// TwinCAT 3 PLC project ContinuousFormulation
// ProgramVersion: 3.1.4020.1
// libraries:
//   VisuElemTextEditor, 3.5.6.0 (System)
//   visuinputs, 3.5.6.0 (system)
//   VisuNativeControl, 3.5.6.0 (System)
//   Tc2_ModbusSrv, * (Beckhoff Automation GmbH)
//   Tc2_SerialCom, * (Beckhoff Automation GmbH)
//   Tc2_Standard, * (Beckhoff Automation GmbH)
//   Tc2_System, * (Beckhoff Automation GmbH)
//   Tc2_SystemCX, * (Beckhoff Automation GmbH)
//   Tc2_Utilities, * (Beckhoff Automation GmbH)
//   Tc3_Interfaces, * (Beckhoff Automation GmbH)
//   Tc3_Module, * (Beckhoff Automation GmbH)
//   VisuDialogs, * (System)
// project tree:
//   DUTs/Wiesler/ ControllerData.TcDUT, elementStatus.TcDUT, FlowCalTestResult.TcDUT, AI.TcDUT, MovingAverage.TcDUT, OLSResult.TcDUT, sAnalogSim.TcDUT, sEU_SCALE.TcDUT, sAnalogConstraint.TcDUT, sWeight.TcDUT, testResults.TcDUT
//   DUTs/Wiesler/Masterflex/ sMasterflexPort.TcDUT
//   / GlobalTextList.TcGTLO, PlcTask.TcTTO
//   GVLs/ Wiesler.TcGVL
//   POUs/FlowCalibration/ FlowCalSequence.TcPOU, OLS.TcPOU, testOLS.TcPOU
//   POUs/ MAIN.TcPOU, MTSerial.TcPOU, sonotecCalibration.TcPOU, FlowCheck.TcPOU, SonotecFreq.TcPOU
//   POUs/Wiesler/ AI1.TcPOU, AO1.TcPOU, fbDatalogger.TcPOU, fbGetUnixTime.TcPOU, fbMovingAverage.TcPOU, FQ1.TcPOU, ModbusTCPReveal.TcPOU, MT_SICS_TO_Weight.TcPOU, randn.TcPOU
//   POUs/Wiesler/DataConversion/ wordArray2Real.TcPOU, wordArray2DINT.TcPOU
//   POUs/Wiesler/Datalog/ fbDatalogger_100ms.TcPOU, fbDatalogger_10ms.TcPOU, fbDatalogger_1ms.TcPOU, fbDatalogger_1s.TcPOU, fbDatalogger_20ms.TcPOU, fShiftArray.TcPOU
//   POUs/Wiesler/FlowConcentrationControl/ CC1.TcPOU, FC2_Preload.TcPOU, FlowSequence_CC1Test.TcPOU, FVC3.TcPOU, StartStopSequence_CC1Test.TcPOU, FV3.TcPOU, testFC.TcPOU (not stored)
//   POUs/Wiesler/Masterflex/ fbMasterflex.TcPOU, fbMasterflexControl.TcPOU, fbMasterflexSerial.TcPOU
//   VISUs/ ContinuousFormulation.TcVIS, HMI.TcVIS, ImagePool.TcIPO (not stored), VisualizationManager.TcVMO (not stored)
// real-time tasks:
//   TASK PlcTask: cycle T#1ms, priority 20, ADS port 350
// I/O:
//   DEVICE Device 1 (EtherCAT), AmsNetId 5.31.160.194.2.1
//     Term 1 (EK1200) [EK1200-5000 EtherCAT Power supply (2A E-Bus)]
//       Term 2 (EL1004) [EL1004 4Ch. Dig. Input 24V, 3ms]
//       Term 3 (EL2004) [EL2004 4Ch. Dig. Output 24V, 0.5A]
//       Term 4 (EL3124) Flow [EL3124 4Ch. Ana. Input 4-20mA Diff.]
//       Term 5 (EL3124) Optek [EL3124 4Ch. Ana. Input 4-20mA Diff.]
//       Term 6 (EL3124) Reveal [EL3124 4Ch. Ana. Input 4-20mA Diff.]
//       Term 7 (EL3124) [EL3124 4Ch. Ana. Input 4-20mA Diff.]
//       Term 8 (EL3104) [EL3104 4Ch. Ana. Input +/-10V Diff.]
//       Term 9 (EL3702) [EL3702 2Ch. Ana. Input +/-10V, DIFF, Oversample]
//       Term 10 (EL4124) [EL4124 4Ch. Ana. Output 4-20mA, 16bit]
//       Term 11 (EL6002) [EL6002 Interface 2Ch. (RS232)]
//       Term 12 (EL6002) [EL6002 Interface 2Ch. (RS232)]
//       Term 13 (EL1502) [EL1502 2Ch. +/- Counter 24V, 100kHz]
//       Term 14 (EL9011) [EL9011 End Terminal]
// variable links:
//   ContinuousFormulation/ContinuousFormulation Instance <-> Device 1 (EtherCAT)/Term 1 (EK1200)/Term 11 (EL6002)
//     PlcTask Inputs/MAIN.P9999A.stIn_Port/D[{0..21}] <-> COM TxPDO-Map Inputs Channel 1/Data In {0..21}  (22 links)
//     PlcTask Inputs/MAIN.P9999A.stIn_Port/Status <-> COM TxPDO-Map Inputs Channel 1/Status
//     PlcTask Inputs/MAIN.P9999B.stIn_Port/D[{0..21}] <-> COM TxPDO-Map Inputs Channel 2/Data In {0..21}  (22 links)
//     PlcTask Inputs/MAIN.P9999B.stIn_Port/Status <-> COM TxPDO-Map Inputs Channel 2/Status
//     PlcTask Outputs/MAIN.P9999A.stOut_Port/Ctrl <-> COM RxPDO-Map Outputs Channel 1/Ctrl
//     PlcTask Outputs/MAIN.P9999A.stOut_Port/D[{0..21}] <-> COM RxPDO-Map Outputs Channel 1/Data Out {0..21}  (22 links)
//     PlcTask Outputs/MAIN.P9999B.stOut_Port/Ctrl <-> COM RxPDO-Map Outputs Channel 2/Ctrl
//     PlcTask Outputs/MAIN.P9999B.stOut_Port/D[{0..21}] <-> COM RxPDO-Map Outputs Channel 2/Data Out {0..21}  (22 links)
//   ContinuousFormulation/ContinuousFormulation Instance <-> Device 1 (EtherCAT)/Term 1 (EK1200)/Term 12 (EL6002)
//     PlcTask Inputs/MTSerial.stIn_Port/D[{0..21}] <-> COM TxPDO-Map Inputs Channel 1/Data In {0..21}  (22 links)
//     PlcTask Inputs/MTSerial.stIn_Port/Status <-> COM TxPDO-Map Inputs Channel 1/Status
//     PlcTask Outputs/MTSerial.stOut_Port/Ctrl <-> COM RxPDO-Map Outputs Channel 1/Ctrl
//     PlcTask Outputs/MTSerial.stOut_Port/D[{0..21}] <-> COM RxPDO-Map Outputs Channel 1/Data Out {0..21}  (22 links)
//   ContinuousFormulation/ContinuousFormulation Instance <-> Device 1 (EtherCAT)/Term 1 (EK1200)/Term 2 (EL1004)
//     PlcTask Inputs/MAIN.AC9999C.lsh <-> Channel 2/Input
//     PlcTask Inputs/MAIN.AC9999C.lsl <-> Channel 1/Input
//   ContinuousFormulation/ContinuousFormulation Instance <-> Device 1 (EtherCAT)/Term 1 (EK1200)/Term 3 (EL2004)
//     PlcTask Outputs/MAIN.FV9999C.activeSV <-> Channel 2/Output
//     PlcTask Outputs/MAIN.FV9999C.passiveSV <-> Channel 1/Output
//   ContinuousFormulation/ContinuousFormulation Instance <-> Device 1 (EtherCAT)/Term 1 (EK1200)/Term 4 (EL3124) Flow
//     PlcTask Inputs/MAIN.FT9999A.raw <-> AI Standard Channel 2/Value
//     PlcTask Inputs/MAIN.FT9999A.status <-> AI Standard Channel 2/Status
//     PlcTask Inputs/MAIN.FT9999B.raw <-> AI Standard Channel 1/Value
//     PlcTask Inputs/MAIN.FT9999B.status <-> AI Standard Channel 1/Status
//     PlcTask Inputs/MAIN.FT9999C.raw <-> AI Standard Channel 3/Value
//     PlcTask Inputs/MAIN.FT9999C.status <-> AI Standard Channel 3/Status
//   ContinuousFormulation/ContinuousFormulation Instance <-> Device 1 (EtherCAT)/Term 1 (EK1200)/Term 6 (EL3124) Reveal
//     PlcTask Inputs/MAIN.AT9999RV{290..320 step 10}.raw <-> AI Standard Channel {1..4}/Value  (4 links)
//     PlcTask Inputs/MAIN.AT9999RV{290..320 step 10}.status <-> AI Standard Channel {1..4}/Status  (4 links)
//   ContinuousFormulation/ContinuousFormulation Instance <-> Device 1 (EtherCAT)/Term 1 (EK1200)/Term 8 (EL3104)
//     PlcTask Inputs/MAIN.AT9999CWx.raw <-> AI Standard Channel 4/Value
//     PlcTask Inputs/MAIN.AT9999CWx.status <-> AI Standard Channel 4/Status
//     PlcTask Inputs/MAIN.PT9999A.raw <-> AI Standard Channel 1/Value
//     PlcTask Inputs/MAIN.PT9999A.status <-> AI Standard Channel 1/Status
//     PlcTask Inputs/MAIN.PT9999B.raw <-> AI Standard Channel 2/Value
//     PlcTask Inputs/MAIN.PT9999B.status <-> AI Standard Channel 2/Status
//     PlcTask Inputs/MAIN.PT9999C.raw <-> AI Standard Channel 3/Value
//     PlcTask Inputs/MAIN.PT9999C.status <-> AI Standard Channel 3/Status
//   ContinuousFormulation/ContinuousFormulation Instance <-> Device 1 (EtherCAT)/Term 1 (EK1200)/Term 9 (EL3702)
//     PlcTask Inputs/MAIN.AT9999CWYY.raw <-> Ch2 Sample 0/Ch2 Value
//     PlcTask Inputs/MAIN.AT9999CWy.raw <-> Ch1 Sample 0/Ch1 Value

CONFIGURATION ContinuousFormulation
    RESOURCE PLC ON TwinCAT3
        TASK PlcTask(INTERVAL := T#1ms, PRIORITY := 20);
        PROGRAM MAIN WITH PlcTask : MAIN;
        PROGRAM FlowCheck WITH PlcTask : FlowCheck;
        PROGRAM StartStopSequence_CC1Test WITH PlcTask : StartStopSequence_CC1Test;
    END_RESOURCE
END_CONFIGURATION

// ---- DUTs/Wiesler/ControllerData.TcDUT
TYPE ControllerData :
STRUCT
	Kp : LREAL := 1.0; //Gain
	Ti : TIME := T#5S; //Integral time
	execTime : TIME := T#500MS; //Time between controller executions
END_STRUCT
END_TYPE

// ---- DUTs/Wiesler/elementStatus.TcDUT
TYPE elementStatus :
(
    Bad := 0,
    Timeout := 1,
	Unknown := 11,
    Good := 12
);
END_TYPE

// ---- DUTs/Wiesler/FlowCalTestResult.TcDUT
TYPE FlowCalTestResult :
STRUCT
	flow : LREAL;
	weight : LREAL;
	startTime : 
END_STRUCT
END_TYPE

// ---- DUTs/Wiesler/Masterflex/sMasterflexPort.TcDUT
TYPE sMasterflexPort :
STRUCT
	// I/O variables for a EL6001 terminal
	stIn_Port AT %I*	: EL6inData22B;	// linked to the EL6002 in the TwinCAT System Manager
	stOut_Port AT %Q*	: EL6outData22B; // linked to the EL6002 in the TwinCAT System Manager
	
	//Serial send variables
	sSendString: STRING(100) := '';

	//Receive variables
	bReceiveTimeout	: BOOL := FALSE;
	sRxSuffix : STRING(5) := '';
	nReceiveCounter	: UDINT := 0;
	sLastReceivedString: STRING(30) := '';
	bListening : BOOL := FALSE;
	tListenTON : TON;
	
	//Pump Status
	fSpeedPV : LREAL := -100.0;
	fFlowPV : LREAL := 0.0;		//Calculated flow in mg/min
	fSpeedSP : LREAL := -100.0;
	fFlowSP : LREAL := -100.0;
	bRun : BOOL := FALSE;
	bLocal : BOOL := FALSE;
	bDirection : BOOL := TRUE; //true is positive/forward, false is negative/backwards
	nPumpStatus : INT := -1; //see http://www.coleparmer.com/Assets/manual_pdfs/07551-20,30.pdf pg 3-33
	nCommStatus : INT := -1;
	
	//Pump Requests
	fSpeedSP_RQ : LREAL := 0.0;
	fFlowSP_RQ : LREAL := -100.0;
	nRun_RQ : INT := 0;  //-1=no RQ, 0=Stop, 1=Run
	nDir_RQ : INT := -1;  //-1=no RQ, 0=Backwards, 1=Forwards //TODO this does no twork correctly probably. Pump must be stopped to change direction
	nLocal_RQ : INT := 1; //-1=no RQ, 0=Remote, 1=Local

	//State Control Information
	nLastState : INT := 1;
	nState : INT := 1;
	
	//Pump Configuration
	//Tube Sizes: 13 (.8mm, 1/32"), 14 (1.6mm, 1/16"), 16 (3.1mm, 1/8"), 
	//			  25 (4.8mm, 3/16"), 17 (6.4mm, 1/4"), 18 (7.9mm, 5/16")
	nTubeSize :INT := 13;		//Tube Number
	nHeads : INT := 2;			//Number of heads
	fPeriodMS : LREAL := 1.0;	//Period between pulses in milliseconds
	
	
END_STRUCT
END_TYPE

// ---- DUTs/Wiesler/AI.TcDUT
TYPE AI :
STRUCT
	// IO variables: status and value
	raw AT %I* : INT;
	status AT %I* : INT;
	// AI scaling and simulation
	scale : sEU_SCALE := (euLo := 0,  euHi := 100.0, eu := 'mg/min');
	sim : sAnalogSim;
	// PV and filtered PV
	pv : LREAL := -1000.0;
	pvfilt : LREAL := -1000.0;
	//Low cutoff 
	loCutEnable : BOOL := FALSE; //low cutoff enable
	loCut : LREAL := 0.0; // if pv is less than this, set pv to 0.0
END_STRUCT
END_TYPE

// ---- DUTs/Wiesler/MovingAverage.TcDUT
TYPE MovingAverage :
STRUCT
	arrSize : UINT := 3000; //Do not change online.
	start : UINT := arrSize - 1;
	vals : ARRAY[0..start] OF LREAL := [arrSize(0.0)];
	size : UINT := 1000;
	in : LREAL;
	out : LREAL;
END_STRUCT
END_TYPE

// ---- DUTs/Wiesler/OLSResult.TcDUT
TYPE OLSResult :
STRUCT
	m : LREAL := 0; // calculated linear regression slope
	b : LREAL := 0; // calculated linear regression intercept
	R2 : LREAL := 0; // R squared
	status : INT := 0; // 0 : OK; >0 : any failure
END_STRUCT
END_TYPE

// ---- DUTs/Wiesler/sAnalogSim.TcDUT
TYPE sAnalogSim :
STRUCT
	simEnable : BOOL := FALSE;
	simValue : LREAL := 0.0;
END_STRUCT
END_TYPE

// ---- DUTs/Wiesler/sEU_SCALE.TcDUT
TYPE sEU_SCALE :
STRUCT
	rawLo: INT := 0;
	rawHi: INT := 32767;
	euLo: LREAL := 0.0;
	euHi: LREAL := 100.0;
	eu: STRING[20] := '%';
END_STRUCT
END_TYPE

// ---- DUTs/Wiesler/sAnalogConstraint.TcDUT
TYPE sAnalogConstraint :
STRUCT
	sp : LREAL := 0.0;  //value to be sent to controller
	rq : LREAL := 0.0;  //request from HMI or calculations
	mn : LREAL := 0.0;  //Minimum value
	mx : LREAL := 0.0;  //Maximum value
END_STRUCT
END_TYPE

// ---- DUTs/Wiesler/sWeight.TcDUT
TYPE sWeight :
STRUCT
	pv : LREAL := -10000.0;
	status : string(15) := 'Invalid';
END_STRUCT
END_TYPE

// ---- DUTs/Wiesler/testResults.TcDUT
TYPE testResults :
STRUCT
	P9999Arpm : LREAL := 0.0;
	P9999Atubing : INT := 0;
	P9999Brpm : LREAL := 0.0;
	P9999Btubing : INT := 0;
	FQ9999A : LREAL := 0.0;
	FQ9999B : LREAL := 0.0;
	FQ9999C : LREAL := 0.0;
	FT9999Aavg : LREAL := 0.0;
	FT9999Bavg : LREAL := 0.0;
	FT9999Cavg : LREAL := 0.0;
END_STRUCT
END_TYPE

// ---- GVLs/Wiesler.TcGVL
VAR_GLOBAL
	unixTime : ULINT;
	FC9999ACtrlData : ControllerData := (Kp := 7.0, Ti := T#500MS, execTime := T#200MS);
	FC9999BCtrlData : ControllerData := (Kp := 0.4, Ti := T#500MS, execTime := T#500MS);
END_VAR

VAR_GLOBAL PERSISTENT
	FT9999A_OLS : OLSResult := (m := 1.0, b := 0.0, R2 := 1.0, status := 0);
	P9999A_OLS : OLSResult := (m := 1.0, b := 0.0, R2 := 1.0, status := 0);
	FT9999B_OLS : OLSResult := (m := 1.0, b := 0.0, R2 := 1.0, status := 0);
	P9999B_OLS : OLSResult := (m := 1.0, b := 0.0, R2 := 1.0, status := 0);
END_VAR

// ---- POUs/MAIN.TcPOU
PROGRAM MAIN

VAR CONSTANT
	SAMPLE_SIZE : INT := 1000;
END_VAR

VAR_INPUT
	logActive : BOOL := FALSE;
	MTSendString : STRING(132) := 'SIR$0D$0A';
	//Pump control
	P9999A : sMasterflexPort := (bDirection := FALSE, nTubeSize := 13);
	P9999B : sMasterflexPort := (bDirection := FALSE, nTubeSize := 16);
	//totalizer blocks
	fbFQ9999A : FQ1;
	fbFQ9999B : FQ1;
	fbFQ9999C : FQ1;
	FQ9999_MasterReset : BOOL; //Master reset - resets all totalizers
	AQ9999C : LREAL; // implied concentration based on FQA and FQB
	
	phase : UINT := 0;
	//Flow and Concentration Control
	FC9999A : FC2_Preload;
	FC9999B : FC2_Preload;
	AC9999C : CC1;
	FV9999C : FV3;
	FVC9999C : FVC3;

END_VAR

VAR
	//test
    Tau : LREAL := 1.0;
	FilterFactor : LREAL;
	ftfirstorder : LREAL;
	//-test
	heartbeat : DINT;
	fbGetUnixTimeGlobal : fbGetUnixTime;
	temp : UINT;
	MTWeight : sWeight;
	
	//Flowmeters
	FT9999A : AI := (loCutEnable:= FALSE, loCut := 0.25, scale := (euLo := -20.0,  euHi := 100.0, eu := 'ml/min')); //E+H small
	FT9999B : AI := (loCutEnable:= TRUE, loCut := 2.25, scale := (euLo := 0,  euHi := 1000.0, eu := 'ml/min')); //E+H large
	FT9999C : AI := (loCutEnable:= TRUE, loCut := 2.25, scale := (euLo := 0,  euHi := 1000.0, eu := 'ml/min')); //E+H very large
	
	//Pressures
	PT9999A : AI := (scale := (euLo := 0,  euHi := 15.0, eu := 'psig'));
	PT9999B : AI := (scale := (euLo := 0,  euHi := 15.0, eu := 'psig'));
	PT9999C : AI := (scale := (euLo := 0,  euHi := 15.0, eu := 'psig'));

	//Reveal
	AT9999RV290 : AI := (scale := (euLo := -0.1,  euHi := 2.0, eu := 'AU'));
	AT9999RV300 : AI := (scale := (euLo := -0.1,  euHi := 1.1, eu := 'mg/ml'));
	AT9999RV310 : AI := (scale := (euLo := 0,  euHi := 2.0, eu := 'AU'));
	AT9999RV320 : AI := (scale := (euLo := 0,  euHi := 2.0, eu := 'AU'));
	AT9999C : ModbusTCPReveal();

	//ColorWise
	AT9999CWx  : AI := (scale := (rawLo := 0, rawHi := 16383, euLo := 0,  euHi := 1.0, eu := 'x'));
	AT9999CWy  : AI := (scale := (rawLo := 0, rawHi := 16383, euLo := 0,  euHi := 1.0, eu := 'y'));
	AT9999CWYY : AI := (scale := (rawLo := 0, rawHi := 16383, euLo := 0,  euHi := 1.0, eu := 'Y'));

	//function blocks
	fbP9999A : fbMasterflex;
	fbP9999B : fbMasterflex;
	
	//Phases
	FT9999A_FLOWCAL : FlowCalSequence;
	FT9999B_FLOWCAL : FlowCalSequence;
	
	//AI blocks
	fbFT9999A : AI1;
	fbFT9999B : AI1;
	fbFT9999C : AI1;
	fbPT9999A : AI1;
	fbPT9999B : AI1;
	fbPT9999C : AI1;
	fbAT9999RV290 : AI1;
	fbAT9999RV300 : AI1;
	fbAT9999RV310 : AI1;
	fbAT9999RV320 : AI1;
	fbAT9999CWx  : AI1;
	fbAT9999CWy  : AI1;
	fbAT9999CWYY : AI1;
	
	// filter blocks
	fbFT9999AFilt : fbMovingAverage;
	FT9999ASize : UINT := 500;
	FT9999AFiltTarget : LREAL := 1500.0; //Target number of ms to for moving average
	fbFT9999BFilt : fbMovingAverage;
	FT9999BSize : UINT := 500;
	FT9999BFiltTarget : LREAL := 1500.0; //Target number of ms to for moving average
	fbFT9999CFilt : fbMovingAverage;
	FT9999CSize : UINT := 500;
	fbFT9999CfqFilt : fbMovingAverage;

	//Data logging
	fbP9999ARPMlog : fbDatalogger_100ms;
	fbP9999AFlowlog : fbDatalogger_100ms;
	fbP9999BRPMlog : fbDatalogger_100ms;
	fbP9999BFlowlog : fbDatalogger_100ms;
		
	fbFT9999Alog : fbDatalogger_1ms;
	fbFT9999Blog : fbDatalogger_1ms;
	fbFT9999Clog : fbDatalogger_1ms;
	
	fbFT9999Afiltlog : fbDatalogger_100ms;
	fbFT9999Bfiltlog : fbDatalogger_100ms;
	fbFT9999Cfiltlog : fbDatalogger_100ms;
	
	fbFQ9999Alog : fbDatalogger_100ms;
	fbFQ9999Blog : fbDatalogger_100ms;
	fbFQ9999Clog : fbDatalogger_100ms;
	
	fbPT9999Alog : fbDatalogger_1ms;
	fbPT9999Blog : fbDatalogger_1ms;
	fbPT9999Clog : fbDatalogger_1ms;

	fbWT9999Clog : fbDatalogger_100ms;

	fbAT9999RV290log : fbDatalogger_10ms;
	fbAT9999RV300log : fbDatalogger_10ms;
	fbAT9999RV310log : fbDatalogger_10ms;
	fbAT9999RV320log : fbDatalogger_10ms;

	fbAT9999CWxlog  : fbDatalogger_1ms;
	fbAT9999CWylog  : fbDatalogger_1ms;
	fbAT9999CWYYlog : fbDatalogger_1ms;
	
END_VAR

heartbeat := heartbeat + 1;
fbGetUnixTimeGlobal();  //set global variable unixTime
//Code that runs 1 time per second
IF (heartbeat MOD 1000) = 0 THEN
	temp := MIN(2499,DINT_TO_UINT(3*TRUNC(P9999A.fPeriodMS)));  //lower bound is 3 * period - want to make sure at least 3 periods are averaged
	FT9999ASize := LIMIT(temp, DINT_TO_UINT((TRUNC(P9999A.fPeriodMS) * TRUNC(FT9999AFiltTarget/P9999A.fPeriodMS))), 2500);
	temp := MIN(2499,DINT_TO_UINT(3*TRUNC(P9999B.fPeriodMS)));  //lower bound is 3 * period - want to make sure at least 3 periods are averaged
	FT9999BSize := LIMIT(temp, DINT_TO_UINT((TRUNC(P9999B.fPeriodMS) * TRUNC(FT9999BFiltTarget/P9999B.fPeriodMS))), 2500);
END_IF

//Call serial line handlers
MTSerial(sSendString := MTSendString, weight := MTWeight);

//Call pump handler
fbP9999A(sPort := P9999A);
fbP9999B(sPort := P9999B);

//Valve handlers
fv9999c();


//Flow transmitters
fbFT9999A(AI := FT9999A);
fbFT9999AFilt(in := FT9999A.pv, size := FT9999ASize, out => FT9999A.pvfilt);

//test
FilterFactor := 1.0 - EXP(-0.001/tau);
ftfirstorder := (1.0 - filterfactor) * ftfirstorder + filterfactor * FT9999A.pv;
//-test


fbFQ9999A(flow := FT9999A.pv, timeBaseMS := (1000.0*60.0));
fbFT9999B(AI := FT9999B);
fbFT9999BFilt(in := FT9999B.pv, size := FT9999BSize, out => FT9999B.pvfilt);
fbFQ9999B(flow := FT9999B.pv, timeBaseMS := (1000.0*60.0));
fbFT9999C(AI := FT9999C);
fbFT9999CFilt(in := FT9999C.pv, size := FT9999CSize, out => FT9999C.pvfilt);
fbFQ9999C(flow := FT9999C.pv, timeBaseMS := (1000.0*60.0));
//reset all totalizers if master reset 
IF FQ9999_MasterReset THEN
	fbFQ9999A.resetRQ := TRUE;
	fbFQ9999B.resetRQ := TRUE;
	fbFQ9999C.resetRQ := TRUE;
	FQ9999_MasterReset := FALSE;
END_IF
//Calculate average concentration
IF (fbFQ9999A.total + fbFQ9999B.total) > 0.0 THEN
	AQ9999C := (fbFQ9999A.total*AC9999C.API_Concentration)/(fbFQ9999A.total + fbFQ9999B.total);
ELSE
	AQ9999C := 0.0;
END_IF

//Flow and Concentration Control
FC9999A(FTOLS := FT9999A_OLS, pumpOLS := P9999A_OLS, pump := P9999A, ft := FT9999A, ctrlData:= FC9999ACtrlData);
FC9999B(FTOLS := FT9999B_OLS, pumpOLS := P9999B_OLS, pump := P9999B, ft := FT9999B, ctrlData:= FC9999BCtrlData);
FT9999A_FLOWCAL(fq := fbFQ9999A, pump := P9999A, FTOLS := FT9999A_OLS, pumpOLS := P9999A_OLS);
FT9999B_FLOWCAL(fq := fbFQ9999B, pump := P9999B, FTOLS := FT9999B_OLS, pumpOLS := P9999B_OLS);
AC9999C(FCA := FC9999A, FTA := FT9999A, FCB:= FC9999B, FTB := FT9999B, PumpA := P9999A, PumpB := P9999B);
FVC9999C(FTA := FT9999A, FTB := FT9999B, ATC := AT9999C, cc := AC9999C, API_Concentration := AC9999C.API_Concentration, FV := FV9999C);

//Pressure
fbPT9999A(AI := PT9999A);
fbPT9999B(AI := PT9999B);
fbPT9999C(AI := PT9999C);

//Reveal
AT9999C();

//ColorWise
fbAT9999CWx(AI := AT9999CWx);
fbAT9999CWy(AI := AT9999CWy);
fbAT9999CWYY(AI := AT9999CWYY);

//Data Logging
fbP9999ARPMlog(fData := P9999A.fSpeedPV);
fbP9999AFlowlog(fData := P9999A.fFlowPV);
fbP9999BRPMlog(fData := P9999B.fSpeedPV);
fbP9999BFlowlog(fData := P9999B.fFlowPV);
	
fbFT9999Alog(fData := FT9999A.pv);;
fbFT9999Blog(fData := FT9999B.pv);
fbFT9999Clog(fData := FT9999C.pv);

fbFT9999Afiltlog(fData := FT9999A.pvfilt);
fbFT9999Bfiltlog(fData := FT9999B.pvfilt);
fbFT9999Cfiltlog(fData := FT9999C.pvfilt);

fbFQ9999Alog(fData := fbFQ9999A.total);
fbFQ9999Blog(fData := fbFQ9999B.total);
fbFQ9999Clog(fData := fbFQ9999C.total);

fbPT9999Alog(fData := PT9999A.pv);
fbPT9999Blog(fData := PT9999B.pv);
fbPT9999Clog(fData := PT9999C.pv);

fbWT9999Clog(fData := MTWeight.pv);

fbAT9999RV290log(fData := AT9999RV290.pv);
fbAT9999RV300log(fData := AT9999RV300.pv);
fbAT9999RV310log(fData := AT9999RV310.pv);
fbAT9999RV320log(fData := AT9999RV320.pv);

fbAT9999CWxlog(fData := AT9999CWx.pv);
fbAT9999CWylog(fData := AT9999CWy.pv);
fbAT9999CWYYlog(fData := AT9999CWYY.pv);

//Phase Control
CASE phase OF
1:
	FT9999A_FLOWCAL.start := TRUE;
	phase := 0;
2:
	FT9999B_FLOWCAL.start := TRUE;
	phase := 0;
END_CASE

END_PROGRAM

// ---- POUs/Wiesler/FQ1.TcPOU
FUNCTION_BLOCK FQ1
VAR_INPUT
	enable : BOOL := TRUE;
	resetRQ : BOOL := FALSE;
	flow : LREAL := 0.0;
	timeBaseMS : LREAL := 1000.0*60.0;
END_VAR
VAR_IN_OUT
END_VAR
VAR_OUTPUT
	total : LREAL := 0.0;
END_VAR
VAR
	scanMS : LREAL := 1.0;
END_VAR

IF resetRQ THEN
	total := 0.0;
	resetRQ := FALSE;
ELSE
	IF enable THEN
		total := total + flow*scanMS/timeBaseMS;		
	END_IF
END_IF

END_FUNCTION_BLOCK

// ---- POUs/Wiesler/FlowConcentrationControl/FC2_Preload.TcPOU
FUNCTION_BLOCK FC2_Preload
VAR_INPUT
	SP : LREAL := 0.0;
	uncalFTPV : LREAL := 0;
	modeSP : UINT := 1; //controller mode Setpoint.  1 is Manual, 2 is Auto
	outMax : LREAL := 600.0;
	outMin : LREAL := 10.0; //don't allow pump speed to go below 10 RPM
	SPMin : LREAL := 1.0; //don't allow SP to be less than 1.0 mL/min
END_VAR
VAR_IN_OUT
	FTOLS : OLSResult;
	pumpOLS : OLSResult;
	pump : sMasterflexPort;
	ft : AI;
	ctrlData : ControllerData;
END_VAR
VAR_OUTPUT

END_VAR
VAR
	PV : LREAL := 0.0;
	outBase : LREAL := 0.0 ; //Base OUT value predicted by flow vs. speed correlation
	OUT : LREAL := 0.0;
	lastOUT: LREAL := 0.0;
	modeAct : UINT := 2; //controller mode Actual.  1 is Manual, 2 is Auto, 3 is Suspend
	lastModeAct : UINT;
	execCounter : DWORD := 0;
	iError : LREAL;
	integral : LREAL;
	integralAtOutMax : LREAL;
	integralAtOutMin : LREAL;
	lastIntegral : LREAL;
	lastSP : LREAL;
	
	fbSuspend : TP;
	newSP : BOOL;
	newPumpOn : BOOL;
	pumpModeOn : BOOL;
	lastPumpModeOn : BOOL;
	suspendTime : TIME := T#2S;
	
END_VAR

//PV := FTOLS.m * ft.pvfilt + FTOLS.b;  //DO NOT scale ft to adjust for zero
PV := ft.pvfilt;
SP := MAX(SP, SPMin);
pumpModeOn := ((NOT pump.bLocal AND pump.bRun));
execCounter := execCounter + 1;

modeAct := modeSP;
//Calculate integration suspend - when SP changes or the mode has just gone to Auto.
newSP := (lastSP <> SP OR (modeAct = 2 AND lastModeAct <> 2));
newPumpOn := (lastPumpModeOn <> pumpModeOn);
IF newSP THEN
	//lastIntegral := lastIntegral * SP/MAX(lastSP, 0.01);
	//lastIntegral := LIMIT(outMin, lastIntegral, outMax);
END_IF
fbSuspend(IN := (newSP OR newPumpOn), PT := suspendTime);

//Control algorithm
IF execCounter >= TIME_TO_DWORD(ctrlData.execTime) THEN
	execCounter := 0;
	//Execute control algorithm
	CASE modeAct OF
		2: //Control is in Auto
			outBase := pumpOLS.m * SP + pumpOLS.b;
			//calculate new integral component unless integration is suspended
			IF fbSuspend.Q OR ((modeSP = 2) AND (pump.bLocal OR NOT pump.bRun)) THEN
				iError := 0.0;
			ELSE
				iError := (SP - PV) * ctrlData.Kp * DWORD_TO_LREAL(TIME_TO_DWORD(ctrlData.execTime))/DWORD_TO_LREAL(TIME_TO_DWORD(ctrlData.Ti));
			END_IF		
			//calculate integral taking into account the ARW and Output min and max
			integralAtOutMax := (outMax - outBase);  //integral value that would make OUT = outMax
			integralAtOutMin := (outMin - outBase);  //integral value that would make OUT = outMin
			integral := MAX(integralAtOutMin, MIN(integralAtOutMax,(lastIntegral + iError)));
			//set output to be the bias calculated by the flow vs. speed correlation and integral action
			OUT := outBase + integral;
			OUT := DINT_TO_LREAL(LREAL_TO_DINT(OUT*10.0))/10.0; //round to tenth
			IF OUT <> lastOut THEN
				pump.fSpeedSP_RQ := OUT;
			END_IF
		1: //Control is in Manual
			integral := 0.0;
			OUT := 0.0;		
	END_CASE
	lastIntegral := integral;
	lastOut := OUT;
END_IF

lastSP := SP;
lastPumpModeOn := pumpModeOn;
lastModeAct := modeAct;

END_FUNCTION_BLOCK

// ---- POUs/Wiesler/FlowConcentrationControl/CC1.TcPOU
FUNCTION_BLOCK CC1
//Concentration Control
//Sets FC Setpoints to achieve target concentration.  At this point no feedback.
VAR_INPUT
	mode : UINT := 0; //0 = manual, 1=Final conc and total flow set directly
	API_Concentration : LREAL := 42.0; //	API Concentration in mg/mL
	conc : sAnalogConstraint := (sp := 0.0, rq := -100.0, mn := 0.0, mx := 1.0);
	a : sAnalogConstraint := (sp := 0.0, rq := -100.0, mn := 2.0, mx := 70.0);
	b : sAnalogConstraint := (sp := 0.0, rq := -100.0, mn := 20.0, mx := 500.0);
	c : sAnalogConstraint := (sp := 0.0, rq := -100.0, mn := 0.0, mx := 500.0);
	lsh AT %I* : BOOL := FALSE;
	lsl AT %I* : BOOL := FALSE;
	autoFill : UINT := 0; //0 = manual (not filling), 1 = auto fill ON
END_VAR
VAR_IN_OUT
	FCA : FC2_Preload;
	FTA : AI;
	FCB : FC2_Preload;
	FTB : AI;
	PumpA : sMasterflexPort;
	PumpB : sMasterflexPort;	
END_VAR
VAR_OUTPUT
END_VAR
VAR
	lastMode : UINT := 0;
	lastAPI_Concentration : LREAL := 42.0;
	filling : BOOL := TRUE;
END_VAR

//Determine constraints on concentration and final flow
c.mx := a.mx + b.mx;
c.mn := 0.0;
conc.mx := API_Concentration;
conc.mn := 0.0;
c.sp := LIMIT(c.mn, c.sp, c.mx);
conc.sp := LIMIT(conc.mn, conc.sp, conc.mx);

//Check of concentration or flow requests are different or filling and pumps OFF
IF c.rq <> c.sp OR conc.rq <> conc.sp OR API_Concentration <> lastAPI_Concentration OR (filling AND (NOT PumpA.bRun AND NOT PumpB.bRun)) THEN
	a.rq := c.rq * conc.rq/MAX(0.0001,API_Concentration);
	b.rq := c.rq - a.rq;
	
	//Check if both flows are in valid ranges
	IF (a.rq = 0.0 OR (a.rq >= a.mn AND a.rq <= a.mx)) AND 
       (b.rq = 0.0 OR (b.rq >= b.mn AND b.rq <= b.mx)) THEN
		a.sp := a.rq;
		b.sp := b.rq;
		c.sp := c.rq;
		conc.sp := conc.rq;
	ELSE
		IF API_Concentration <> lastAPI_Concentration THEN //API concetration changed outside acceptable range.  Go to manual
			mode := 0;
		END_IF
		c.rq := c.sp;
		conc.rq := conc.sp;		
	END_IF
END_IF

// check level
IF NOT lsl THEN
	filling := TRUE;
END_IF
IF lsh THEN
	filling := FALSE;
END_IF

IF NOT filling AND autoFill = 1 THEN // if we are NOT filling (and in autoFill mode) then turn off pumps
	a.sp := 0;
	b.sp := 0;
END_IF

//set flow control setpoint and pump on/off command for API and buffer (both have to be on or both off)
//drive pumps and speed setpoints
IF mode = 1 AND (lastMode <> 1 OR ((PumpA.bLocal = TRUE OR PumpB.bLocal=TRUE) AND filling)) THEN
	PumpA.nLocal_RQ := 0;
	PumpB.nLocal_RQ := 0;
END_IF
IF mode = 1 THEN  //only set flow rates and pump states if in Auto and filling (Not discharging)
	//turn on or off pump A
	IF a.sp >= a.mn THEN
		FCA.modeSP := 2; //auto
		FCA.SP := a.sp;
		IF NOT PumpA.bRun THEN
			PumpA.nRun_RQ := 1;
		END_IF
	ELSE
		FCA.modeSP := 1; //manual
		IF PumpA.bRun THEN
			PumpA.nRun_RQ := 0;
		END_IF
	END_IF
	//turn on or off pump B
	IF b.sp >= b.mn THEN 
		FCB.modeSP := 2; //auto
		FCB.SP := b.sp;
		IF NOT PumpB.bRun THEN
			PumpB.nRun_RQ := 1;
		END_IF
	ELSE
		FCB.SP := b.mn;
		IF PumpB.bRun THEN
			PumpB.nRun_RQ := 0;
		END_IF
	END_IF
END_IF
//if mode has transitioned to 0 (manual) turn off pumps.
IF mode = 0  AND lastMode <> 0 THEN
	FCA.modeSP := 1; //manual
	IF PumpA.bRun THEN
		PumpA.nRun_RQ := 0;
	END_IF
	FCA.SP := b.mn;
	IF PumpB.bRun THEN
		PumpB.nRun_RQ := 0;
	END_IF	
END_IF
lastMode := mode;
lastAPI_Concentration := API_Concentration;

END_FUNCTION_BLOCK

// ---- POUs/Wiesler/FlowConcentrationControl/FV3.TcPOU
// Implementation of a pseudo 3-way valve by controlling 2 outputs 
FUNCTION_BLOCK FV3
VAR_INPUT
	sp : BOOL := FALSE;
END_VAR
VAR_OUTPUT
	pv : BOOL := FALSE;
END_VAR
VAR
	passiveSV AT %Q*: BOOL;
	activeSV AT %Q*: BOOL;
END_VAR

passiveSV := NOT sp;
activeSV := sp;
pv := sp;

END_FUNCTION_BLOCK

// ---- POUs/Wiesler/FlowConcentrationControl/FVC3.TcPOU
FUNCTION_BLOCK FVC3

VAR_INPUT
	mode : UINT := 0; // 0 = manual, 1 = valve controlled by conc spec
	FTA : AI; 
	FTB : AI;
	ATC : ModbusTCPReveal();
	cc : CC1;
	scanMS : LREAL := 1.0;  // number of milliseconds per scan of this module
	timeBaseMS : LREAL := 1000.0*60.0; // time base in milliseconds of the flow measurement.  Like mL/min timebase is minutes, so 60*1000 milliseconds
	API_Concentration : LREAL := 42.0; // mg/mL
END_VAR
VAR_IN_OUT
	FV : FV3;
END_VAR
VAR_OUTPUT
END_VAR
VAR CONSTANT
	nPoints : DINT := 200;
END_VAR
VAR
	//Variables for calculating when new concentration element has been created
	FQAscan : LREAL := 0.0;
	FQBscan : LREAL := 0.0;
	FQA: LREAL := 0.0;
	FQB: LREAL := 0.0;
	FQAscanAdd : LREAL := 0.0;
	FQBscanAdd : LREAL := 0.0;
	temp : LREAL := 0.0;
	
	//Setup geometry and element size
	elementMass : LREAL := 0.5;  //Each element has this amount in grams - change here may require arrays to be bigger
	massBeforePAT : LREAL := 23.0;  //calculated based on current tubing geometry
	PATelement : INT; //element number for PAT
	massBeforeDivert : LREAL := 31.0;
	divertElement : INT; //element number for diversion tee

	//Defaults
	PATConcDefault : LREAL := -100.0;
	PATCountDefault : UINT := 0;
	PATVarianceDefault : LREAL := 0.0;
	elementConcentration : LREAL := -100.0;
	PATTimeDefault : ULINT := 0;
	elStatusDefault : elementStatus := Bad;
	
	//arrays
	mixTime : ARRAY[0..nPoints] OF ULINT;
	rawConc : ARRAY[0..nPoints] OF LREAL; //calculated raw concentration - from API and Buffer conc/flow at mixing tee
	modeledConc : ARRAY[0..nPoints] OF LREAL; //Adjusted conc with mixing effects from laminar flow and back mixer
	PATConc : ARRAY[0..nPoints] OF LREAL; //Average of unique PAT results for the element in the flow cell
	PATCount : ARRAY[0..nPoints] OF UINT; //Count of unique PAT results for the element in the flow cell
	PATVariance : ARRAY[0..nPoints] OF LREAL; //Variance of unique PAT results for the element in the flow cell
		// Get stdev from variance via sqrt(variance/count) or sqrt(variance/(count-1))
	PATTime : ARRAY[0..nPoints] OF ULINT;
	elStatus : ARRAY[0..nPoints] OF elementStatus;
	
	//values to determine in spec or out of spec
	concSpecHi : LREAL := 0.1; // in spec hi limit is concentration control setpoint + this value
	concSpecLo : LREAL := 0.1; // in spec lo limit is concentration control setpoint - this value
	
	//variable to track diversion logic
	divert : BOOL := TRUE;
	
	//value to determine if PAT reading is new
	lastReadingID : DINT := 0;
	lastElStatus : elementStatus := Bad;
	PATtimeoutTime : TIME := T#100MS;
	fbPATtimeout : TON; //timer for determing timeout of PAT
	
	//local variable
	i : INT := 0;
	firstElementTimeMS : ULINT;  //used on network logic to subscribe to changes in arrays
	lastPATConcAverage: LREAL;
	
END_VAR

PATelement := LREAL_TO_INT(massBeforePAT/elementMass);  //PAT element in array
divertElement := LREAL_TO_INT(massBeforeDivert/elementMass);  //Divert tee element in array

// check for new PAT reading
fbPATtimeout(IN := (lastReadingID = ATC.readingID), PT := PATtimeoutTime);

IF lastReadingID <> ATC.readingID THEN
	//calculate running average and variance:
	// http://dsp.stackexchange.com/questions/811/determining-the-mean-and-standard-deviation-in-real-time
	IF PATCount[PATelement] < 1 THEN
		PATConc[PATelement] := 0.0; //if no measurements yet set previous concentration to 0
	END_IF
	lastPATConcAverage := PATConc[PATelement];                                                         //prev_mean
	PATCount[PATelement] := PATCount[PATelement] + 1;                      							   //n
	PATConc[PATelement] := lastPATConcAverage + (ATC.pv - lastPATConcAverage)/PATCount[PATelement];    //m
	PATVariance[PATelement] := PATVariance[PATelement] + (ATC.pv - PATConc[PATelement]) * (ATC.pv - lastPATConcAverage); //S
	// where S = n * variance .... http://people.ds.cam.ac.uk/fanf2/hermes/doc/antiforgery/stats.pdf
	PATTime[PATelement] := unixTime;
END_IF

// integrate flow transmitter values.
FQAscan := FTA.pv*scanMS/timeBaseMS;
FQBscan := FTB.pv*scanMS/timeBaseMS;
temp := FQA + FQB + FQAscan + FQBscan;

//if new flow makes the incoming element large enough, capture a flow element, shift the arrays, execute concentration modeling and control system
IF (temp >= elementMass) THEN
	// determine how much of new API and buffer flow should be added
	temp := elementMass - FQA - FQB;  //amount of element added this scan
	FQAscanAdd := FQAscan * temp / (FQAscan + FQBscan);
	FQBscanAdd := FQBScan * temp / (FQAscan + FQBscan);
	
	FQA := FQA + FQAscanAdd;
	FQB := FQB + FQBscanAdd;
	elementConcentration := API_concentration*FQA/(FQA + FQB);
	
	//Set current element status.  If PAT has timed out, set status to Timeout.
	IF fbPATtimeout.Q THEN  //no update from PAT within timeout time
		elStatus[PATelement] := Timeout;
		lastElStatus := Timeout;
	ELSIF PATCount[PATelement] = 0 THEN //no PAT update for this element, but PAT has not timedout
		IF lastElStatus = Good THEN
			elStatus[PATelement] := Unknown;  //if last PAT result was good, set this to unknown
		ELSE
			elStatus[PATelement] := lastElStatus; //otherwise, set it to Timeout or Bad to make sure unchecked elements are failsafe
		END_IF
	ELSIF PATConc[PATelement] > (cc.conc.sp - concSpecLo) AND PATConc[PATelement] < (cc.conc.sp + concSpecHi) THEN //within spec
		elStatus[PATelement] := Good;
		lastElStatus := Good;
	ELSE //otherwise mark as bad
		elStatus[PATelement] := Bad;
		lastElStatus := Bad;
	END_IF
	
	// shift arrays & initialize new element
	fShiftArray(sizeofArrayElement := SIZEOF(unixTime), pInsertedElement := ADR(unixTime),
				sizeofArray := SIZEOF(mixTime), pArray := ADR(mixTime));
	fShiftArray(sizeofArrayElement := SIZEOF(elementConcentration), pInsertedElement := ADR(elementConcentration),
				sizeofArray := SIZEOF(rawConc), pArray := ADR(rawConc));
	fShiftArray(sizeofArrayElement := SIZEOF(elementConcentration), pInsertedElement := ADR(elementConcentration),
				sizeofArray := SIZEOF(modeledConc), pArray := ADR(modeledConc)); //Change this when modeling
	fShiftArray(sizeofArrayElement := SIZEOF(PATConcDefault), pInsertedElement := ADR(PATConcDefault),
				sizeofArray := SIZEOF(PATConc), pArray := ADR(PATConc));
	fShiftArray(sizeofArrayElement := SIZEOF(PATCountDefault), pInsertedElement := ADR(PATCountDefault),
				sizeofArray := SIZEOF(PATCount), pArray := ADR(PATCount));
	fShiftArray(sizeofArrayElement := SIZEOF(PATVarianceDefault), pInsertedElement := ADR(PATVarianceDefault),
				sizeofArray := SIZEOF(PATVariance), pArray := ADR(PATVariance));
	fShiftArray(sizeofArrayElement := SIZEOF(PATTimeDefault), pInsertedElement := ADR(PATTimeDefault),
				sizeofArray := SIZEOF(PATTime), pArray := ADR(PATTime));
	fShiftArray(sizeofArrayElement := SIZEOF(elStatusDefault), pInsertedElement := ADR(elStatusDefault),
				sizeofArray := SIZEOF(elStatus), pArray := ADR(elStatus));
	firstElementTimeMS := unixTime;
	
	//Determine divert status
	divert := FALSE;
	FOR i := (PATelement + 1) TO divertElement BY 1 DO
		IF elStatus[i] = Bad OR elStatus[i] = Timeout THEN
			divert := TRUE;
		END_IF
	END_FOR

	FQA := FQAscan - FQAscanAdd; //retain the remainder in FQA and FQB
	FQB := FQBscan - FQBscanAdd;
ELSE 
	// not enough for new element so continue to accumulate flows
	FQA := FQA + FQAscan;
	FQB := FQB + FQBscan;
END_IF

//control valve position if in auto
IF mode = 1 THEN
	FV.sp := NOT divert; // waste: false; filler: true
END_IF

//Update last values
lastReadingID := ATC.readingID;

END_FUNCTION_BLOCK

// ---- POUs/Wiesler/ModbusTCPReveal.TcPOU
FUNCTION_BLOCK ModbusTCPReveal
VAR_INPUT
	IPAddress : STRING(15) := '192.168.2.252'; // IP address of modbus server/field device
	modbusTCPPort : UINT := MODBUS_TCP_PORT; // ModbusTCP port, generally port 
    statusReadMS : UINT := 5000; // Number of milliseconds between status reads
   
END_VAR
VAR_OUTPUT
	fbRead : FB_MBReadRegs;
    //settings for reading register blocks, status and results
	simulateEnable : BOOL := FALSE; //enable simulation - randomly calculates PV, no modbus scanning
    statusRead : BOOL := FALSE; //true when reading the status block of data, registers 1-14
	numRegistersStatus : WORD := 14; //number of Modbus 16-bit registers in status read
	startAddressStatus : WORD := 0; //Starting address for status read - 0 corresponds to register 1
	returnDataStatus : ARRAY [1..14] OF WORD; //raw 16-bit results from status read
	numRegistersResults : WORD := 28; //number of Modbus 16-bit registers in results read
	startAddressRes : WORD := 100; //Starting address for results read - 100 corresponds to register 101
	returnDataResults : ARRAY [1..28] OF WORD; //raw 16-bit results from results read

    //converted values from register reads
	heartbeat : INT; //register 1
	revisionNumber : INT; //register 2
    serialNumber : DINT; //register 3-4
	status : INT; //register 5
	lampState : BOOL; //register 6
	samplingState : BOOL; //register 7
    systemHours : REAL; //register 8-9
    lampHours : REAL; //register 10-11
	temperature : REAL; //register 12-13
    activeMethod : INT; //register 14
	readingID : DINT := 0; //register 101-102 NOTE: not currently implemented
    numResults : INT; //register 103
	results : ARRAY [1..12] OF REAL; //registers 104-127
    resultAlarms : INT; //register 128
	pv : LREAL := -1.0;
	samplesCount : DINT := -1;
END_VAR
VAR
	i : UINT;
	j : UINT;
	is : UINT;
	ie : UINT;
	busyLast : BOOL := FALSE;
	busyCounter : UINT := 0;
	pollCount : ULINT := 0;
	lastPollTime : UINT := 0;
	sampleCountTimeMS : ULINT := 1000;
	lastReadingID : DINT := 0;
	newReading : BOOL := FALSE;
	lastReturnDataResults : ARRAY [1..24] OF WORD;
    nextStatusReadTime : ULINT := 0;

	simulate_execCounter  : DWORD := 0;
	simulate_execTime : TIME := T#20MS;  //simulate a new reading this amount of time
	simulate_x1 : DRAND;
	simulate_x2 : DRAND;
	simulate_mean : LREAL := 3.25;
	simulate_sigma : LREAL := 0.1;
	simulate_seed1 : INT;
	simulate_seed2 : INT;
END_VAR


// - Register(s)     Command             Type   Format
// - -------------   ------------------- -----  ------------------------------------------------------------------------
// -    1            Heartbeat            OUT   16-bit integer: continually increasing value every second
// -    2            Revision Number      OUT   16-bit integer: Identifies the format of all following data. Equals “1” for this version.
// -    3 -    4     Serial Number        OUT   32-bit integer: Serial number of the Reveal
// -    5            Status               OUT   16-bit integer: okay=0, anything else indicates an error condition
// -    6            Lamp State           OUT   16-bit integer: 0=off, 1=on
// -    7            Sampling State       OUT   16-bit integer: 0=off, 1=on
// -    8 -    9     System Hours         OUT   32-bit floating point: Number of hours the system has been on
// -   10 -   11     Lamp Hours           OUT   32-bit floating point: Number of hours the lamp has been on
// -   12 -   13     Air Temperature      OUT   32-bit floating point: Temperature inside Reveal chassis, deg C
// -   14            Active Method Number OUT   16-bit integer: TBD
// -   15 -  100     Not Used
// -  101 -  102     Reading ID           OUT   32-bit integer: reading identifier
// -  103            Num Results          OUT   16-bit integer: Number of results in current model.
// -  104 -  105     Result01             OUT   32-bit floating point
// -  106 -  107     Result02             OUT   32-bit floating point
// -  108 -  109     Result03             OUT   32-bit floating point
// -  110 -  111     Result04             OUT   32-bit floating point
// -  112 -  113     Result05             OUT   32-bit floating point
// -  114 -  115     Result06             OUT   32-bit floating point
// -  116 -  117     Result07             OUT   32-bit floating point
// -  118 -  119     Result08             OUT   32-bit floating point
// -  120 -  121     Result09             OUT   32-bit floating point
// -  122 -  123     Result10             OUT   32-bit floating point
// -  124 -  125     Result11             OUT   32-bit floating point
// -  126 -  127     Result12             OUT   32-bit floating point
// -  128            Result Alarms        OUT   16-bit integer: TBD
//
// Notes
// ---------------------------------------------------------------------------------------------------------------------
//  Modbus register and coil reference numbers start with "1", which corresponds to data at offset "0".

// Program uses a single FB_MBReadRegs function block to read either the status registers 1-14 or the
// results registers 101-128.  The status read occurs as base don input statusReadMS, defaulted to 5 seconds.
// Results reads are read repeatedly except when status reads interrupt.
// FB_MB_ReadRegs inputs (from Twincat manual):
//       sIPAddr: Is a string containing the IP address of the target device.
//       nTCPPort: Port number of the target device.
//       nUnitID:   Identification number of a serial sub-network device. If a device is addressed directly via TCP/IP, this 
//                   value must be 16#FF.
//       nQuantity: Number of output registers (data words) to be read. The value of nQuantity must be > 0.
//       nMBAddr: Start address of the output registers to be read (word offset).
//       cbLength: Contains the max. byte size of the destination buffer. The minimum buffer byte size must be: nQuantity * 2.
//       pDestAddr: Contains the address of the destination buffer into which the data are to be read. The buffer can be
//                  a single variable, an array or a structure, whose address can be found with the ADR operator.
//       bExecute: The function block is activated by a rising edge at this input.
//       tTimeout: States the length of the timeout that may not be exceeded by execution of the ADS command.



IF NOT simulateEnable THEN
    IF unixTime > nextStatusReadTime THEN
      statusRead := TRUE;
    END_IF
	IF statusRead THEN //set modbus read request to get status information
		fbRead(sIPAddr := IPAddress,
				nQuantity := numRegistersStatus,
				nMBAddr := startAddressStatus,
				cbLength := SIZEOF(returnDataStatus),
				pDestAddr := ADR(returnDataStatus),
                tTimeout := T#500MS
		);
	ELSE  //otherwise get results data
		fbRead(sIPAddr := IPAddress,
				nQuantity := numRegistersResults,
				nMBAddr := startAddressRes,
				cbLength := SIZEOF(returnDataResults),
				pDestAddr := ADR(returnDataResults),
                tTimeout := T#500MS
		);
	END_IF
    IF fbRead.bBusy THEN //modbus read is in progress, capture read time and reset read request
        busyCounter := busyCounter + 1;
        fbRead.bExecute := FALSE;
    END_IF

	//If modbus request finished since last scan process the data
	IF NOT fbRead.bBusy AND busyLast THEN
		//Capture poll statistics
		pollCount := pollCount + 1;
		lastPollTime := busyCounter;
		busyCounter := 0;

        //Set output variables based on return registers
      	IF statusRead THEN // Set status values if return data are the status registers
         	IF NOT fbRead.bError THEN
				heartbeat := WORD_TO_INT(returnDataStatus[1]);
				revisionNumber := WORD_TO_INT(returnDataStatus[2]);
				serialNumber := wordArray2DINT(returnDataStatus[3], returnDataStatus[4]);
				status := WORD_TO_INT(returnDataStatus[5]);
				lampState := WORD_TO_BOOL(returnDataStatus[6]);
				samplingState := WORD_TO_BOOL(returnDataStatus[7]);
				systemHours := wordArray2Real(returnDataStatus[8], returnDataStatus[9]);
				lampHours := wordArray2Real(returnDataStatus[10], returnDataStatus[11]);
				temperature := wordArray2Real(returnDataStatus[12], returnDataStatus[13]);
				activeMethod := WORD_TO_INT(returnDataStatus[5]);
         	ELSE
				heartbeat := -100;
				status := -100;
         	END_IF
			//set time for next status read
			nextStatusReadTime := unixTime + statusReadMS;
			statusRead := false;
      	ELSE // most recent read was for results
         	//REGISTERS 101-102
			//readingID := wordArray2DINT(returnDataResults[1], returnDataResults[2]);
			//NOTE: the following is a kludge to overcome Reveal bug where readingID is never updated over Modbus
			newReading := FALSE;
			FOR j := 1 TO 24 DO
				IF returnDataResults[j+3] <> lastReturnDataResults[j] THEN
					newReading := TRUE;  //new reading is indicated by any of the return data being different from the last scan
				END_IF
				lastReturnDataResults[j] := returnDataResults[j+3];
			END_FOR
			//increment readingID if new value was read
			IF newReading THEN
				readingID := readingID + 1;
			END_IF
         	//REGISTER 103
         	numResults := WORD_TO_INT(returnDataResults[3]);
         	//REGISTERS 104-127
			FOR i := 1 TO 12 DO
				is := 2*i+2;
				ie := 2*i+3;
				IF NOT fbRead.bError AND samplingState AND status = 0 THEN
				   results[i] := wordArray2Real(returnDataResults[is], returnDataResults[ie]);
				ELSE
				   results[i] := -100.0;
				END_IF
			END_FOR
			//REGISTER 128
			resultAlarms := WORD_TO_INT(returnDataResults[28]); 
         
         	//Set PV based on results
			IF results[7] <= 0.25 THEN
				pv := results[7]; //low concentration model
			ELSE
				pv := results[6]; //high concentration model
			END_IF
      	END_IF
	END_IF


//Ignore the last stuff and simulate a reading if simulateEnable is active
ELSE //simulate is enabled
	IF simulate_execCounter >= TIME_TO_DWORD(simulate_execTime) THEN  //update pv
		simulate_execCounter := 0;
		readingID := readingID + 1;
		//calculate semi-random pv
		simulate_seed1 := ULINT_TO_INT(unixTime);
		simulate_seed2 := simulate_seed1 + 1;
		simulate_x1(Seed := simulate_seed1);
		simulate_x2(Seed := simulate_seed2);
		pv := randn(x1 := simulate_x1.Num, x2 := simulate_x2.Num, mean := simulate_mean, sigma := simulate_sigma);
	END_IF
	simulate_execCounter := simulate_execCounter + 1;
END_IF


//Count the spectrometer reads
IF (unixTime MOD sampleCountTimeMS) = 0 THEN
	samplesCount := readingID - lastReadingID;
	lastReadingID := readingID;
END_IF

//intitiate the next scan
IF NOT fbRead.bBusy AND NOT busyLast AND NOT simulateEnable THEN
	fbRead.bExecute := TRUE;
END_IF

busyLast := fbRead.bBusy;

END_FUNCTION_BLOCK

// ---- POUs/Wiesler/DataConversion/wordArray2DINT.TcPOU
FUNCTION wordArray2DINT : DINT
VAR_INPUT
	wordLeft : WORD;
	wordRight : WORD; 
END_VAR
VAR
	wordArray : ARRAY [1..2] OF WORD;
	ptdint : POINTER TO DINT;
END_VAR

wordArray[2] := wordLeft;
wordArray[1] := wordRight;
ptdint := ADR(wordArray[1]);
wordArray2DINT := ptdint^;

END_FUNCTION

// ---- POUs/Wiesler/DataConversion/wordArray2Real.TcPOU
FUNCTION wordArray2Real : REAL
VAR_INPUT
	wordLeft : WORD;
	wordRight : WORD; 
END_VAR
VAR
	wordArray : ARRAY [1..2] OF WORD;
	ptReal : POINTER TO REAL;
END_VAR

wordArray[2] := wordLeft;
wordArray[1] := wordRight;
ptReal := ADR(wordArray[1]);
wordArray2Real := ptReal^;

END_FUNCTION

// ---- POUs/Wiesler/randn.TcPOU
FUNCTION randn : lreal
VAR_INPUT
	x1 : LREAL;
	x2 : LREAL;
	mean : LREAL := 0.0;
	sigma : LREAL := 1.0;
END_VAR
VAR
	y : LREAL;
END_VAR

//http://www.design.caltech.edu/erik/Misc/Gaussian.html
x1 := limit(0.01, x1, 1.0); //make sure x1 never is close enough to 0 to fault the LN function
y := SQRT(-2.0 * LN(x1)) * COS(2.0 * PI * x2);
randn := (y * sigma) + mean;

END_FUNCTION

// ---- POUs/Wiesler/Datalog/fShiftArray.TcPOU
FUNCTION fShiftArray : BOOL
VAR_INPUT
	sizeofArrayElement : UDINT; // size of datatype in array (count of bytes)
	pInsertedElement : POINTER TO BYTE; // new data
	
	sizeofArray : UDINT; // size of array
	pArray : POINTER TO BYTE; // start of array
END_VAR
VAR
END_VAR

//Shifts all elements of an array up one index, then inserts new data into 1st element
//Top element of array is overwritten

//Move elements 1 through (n-1) into 2 through n
MemMove(destAddr := (pArray + sizeofArrayElement), srcAddr := pArray, n := (sizeofArray - sizeofArrayElement));

//Move new element into first spot of array
MemMove(destAddr := pArray, srcAddr := pInsertedElement, n := sizeofArrayElement);

//Old FW_MemMove command - cannot find documentation about htis version of the command.
//FW_MemMove(pDest := pArray + sizeofArrayElement, pSrc := pArray, cbLen := sizeofArray - sizeofArrayElement);
//FW_MemMove(pDest := pArray, pSrc := pInsertedElement, cbLen := sizeofArrayElement);

END_FUNCTION

// ---- POUs/Wiesler/fbGetUnixTime.TcPOU
FUNCTION_BLOCK fbGetUnixTime
VAR_INPUT
END_VAR
VAR_OUTPUT
END_VAR
VAR
    fbSystemTime : GETSYSTEMTIME;
    timeAsFileTime : T_FILETIME;
    timeAsSystemTime : TIMESTRUCT;
	timeAsDT : DT;
	timeAsULINT : ULINT;	
	
END_VAR

fbSystemTime(timeLoDW=>timeAsFileTime.dwLowDateTime, timeHiDW=>timeAsFileTime.dwHighDateTime);
timeAsSystemTime := FILETIME_TO_SYSTEMTIME(timeAsFileTime); //to get milliseconds
timeAsDT := FILETIME_TO_DT( timeAsFileTime );  //DT is only seconds, no MS component
unixTime := DT_TO_ULINT(timeAsDT) * 1000 + timeAsSystemTime.wMilliseconds; //global variable

END_FUNCTION_BLOCK

// ---- POUs/Wiesler/Masterflex/fbMasterflex.TcPOU
FUNCTION_BLOCK fbMasterflex
VAR_INPUT
END_VAR
VAR_OUTPUT
END_VAR
VAR
	//Pump control
	fbPumpControl : fbMasterflexControl;
	lastPeriodMS : LREAL := 1.0;
END_VAR

VAR_IN_OUT
	sPort : sMasterflexPort;
END_VAR

//Call pump serial port handler
fbPumpControl(sPort := sPort);

//Calculate derived values
IF sPort.fSpeedPV >= 0.1 THEN
	sPort.fPeriodMS := 60000.0/INT_TO_LREAL(sPort.nHeads)/4.0/sPort.fSpeedPV;
ELSE
	sPort.fPeriodMS := MIN(lastPeriodMS, 1.0); //avoid divide by zero
END_IF

lastPeriodMS := sPort.fPeriodMS;

END_FUNCTION_BLOCK

// ---- POUs/Wiesler/Masterflex/fbMasterflexControl.TcPOU
FUNCTION_BLOCK fbMasterflexControl
VAR_INPUT
END_VAR
VAR_OUTPUT
END_VAR
VAR
	bReqTx : BOOL := TRUE;
	fbMFSerial : fbMasterflexSerial;
	nLastReceiveCounter : UDINT := 0;
	n : INT := -1;	
END_VAR

VAR_IN_OUT
	sPort : sMasterflexPort;
END_VAR

//Execute the timeout timer
sPort.tListenTON(in:=sPort.bListening, pt:=T#1S);

//debug
//sPort.dbg1 := 1;
//sPort.dbg2 := SEL(sPort.dbg1 = 1, 10, 20);

//Send the appropriate message based on the state
IF bReqTX THEN
	bReqTx := FALSE;
    sPort.bListening := TRUE;
	CASE sPort.nState OF
	1: //Unconfigured
		sPort.sRxSuffix := '$0D'; // expected response <STX>P?0<CR>
		sPort.sSendString := '$05'; // <ENQ>
	2: //Set Address - Always '01'
		sPort.sRxSuffix := '$06'; // expected response <ACK>
		sPort.sSendString := '$02P01$0D'; // <STX>P01<CR>
	3: //Get Pump Drive Status - Command I
		sPort.sRxSuffix := '$0D'; // expected response <STX>P01Ixxxxx<CR>
		sPort.sSendString := '$02P01I$0D'; // <STX>P01I<CR>
	4: //Check Front Panel Switches - Command K
		sPort.sRxSuffix := '$0D'; // expected response <STX>Kx<CR>
		sPort.sSendString := '$02P01K$0D'; // <STX>P01K<CR>
	5: //Reset Front Panel Switches
		sPort.sRxSuffix := ''; // No expected response
		sPort.sSendString := '$06P01$0D'; // <ACK>P01<CR>
	6: //Request current speed
		sPort.sRxSuffix := '$0D'; // Expected response <STX>S+nnnn.n<CR>
		sPort.sSendString := '$02P01S$0D'; // <STX>P01S<CR>
	7: //Set speed
		sPort.sRxSuffix := '$06'; // expected response <ACK>
		IF (sPort.fSpeedSP_RQ >= 0.0) THEN
			sPort.fSpeedSP := sPort.fSpeedSP_RQ;
		END_IF
		sPort.fSpeedSP_RQ := -100.0;		
		sPort.sSendString := concat('$02P01S', SEL(sPort.bDirection, '-', '+')); 
		sPort.sSendString := concat(sPort.sSendString, LREAL_TO_FMTSTR(sPort.fSpeedSP,1,TRUE)); 
		sPort.sSendString := concat(sPort.sSendString, '$0D'); // <STX>P01S+nnn.n<CR>
	8: //Start or Stop Pump
		sPort.sRxSuffix := '$06'; // expected response <ACK>
		IF sPort.nRun_RQ = 1 THEN
			sPort.sSendString := '$02P01G0$0D'; // <STX>P01G0<CR>
		ELSE 
			sPort.sSendString := '$02P01H$0D'; // <STX>P01H<CR>
		END_IF
		sPort.nRun_RQ := -1;
	10: //Remote - pump always stops when switching between local and remote, either way
		sPort.sRxSuffix := '$06$06'; // expected response <ACK><ACK>
		sPort.sSendString := '$02P01R$0D$02P01H$0D'; // <STX>P01R<CR><STX>P01H<CR>
		sPort.nLocal_RQ := -1;		
	11: //Local
		sPort.sRxSuffix := '$06$06'; // expected response <ACK><ACK>
      	sPort.sSendString := '$02P01H$0D$02P01L$0D'; // <STX>P01H<CR><STX>P01L<CR>
		sPort.nLocal_RQ := -1;		
	END_CASE
END_IF

//Check the serial port
fbMFSerial(sPort := sPort);

//Handle received messages
IF (len(sPort.sSendString) = 0) AND 
         ((nLastReceiveCounter <> sPort.nReceiveCounter) OR sPort.tListenTON.Q OR sPort.nState = 5) THEN
	bReqTX := TRUE; //Set request to send next message
	//if receive timed out, go to state 1 EXCEPT when in state 1 - then try to assume pump is numbered
	//   NOTE: manual says ENQ is the same as I command for numbered pump - NOT TRUE.  
	//        A previously numbered pump will NOT RESPOND to ENQ.
	IF sPort.tListenTON.Q = TRUE THEN //no valid message was received so RX timed out
		IF sPort.nState = 1 THEN
			sPort.nState := 3;
		ELSE
			sPort.nState := 1;
		END_IF
	ELSE  //a valid message was received and needs to be processed
		nLastReceiveCounter := sPort.nReceiveCounter;
		CASE sPort.nState OF
		1: //Received message should be <STX>P?0<CR>
			IF sPort.sLastReceivedString = '$02P?0$0D' THEN
				//set next state
				sPort.nState := 2;
			ELSIF left(sPort.sLastReceivedString,5) = '$02P01I' THEN
				//If pump already has address, ENQ is same as I command
				sPort.nState := 3;
			ELSE
				sPort.nState := -1;  //place holder for action on failure
			END_IF;
		2: //Received message should be <ACK>
			IF sPort.sLastReceivedString = '$06' THEN
				//set next state
				sPort.nState := 3;
			ELSE
				sPort.nState := -2;  //place holder for action on failure
			END_IF
		3: //Received message should be <STX>P01Ixxxxx<CR>
			IF left(sPort.sLastReceivedString,5) = '$02P01I' THEN
				sPort.bLocal := SEL((mid(sPort.sLastReceivedString,1,6) = '0'), FALSE, TRUE); //0 is local
				sPort.bRun := SEL((mid(sPort.sLastReceivedString,1,9) = '3'), FALSE, TRUE); //3 is pump running
				sPort.nPumpStatus := STRING_TO_INT(mid(sPort.sLastReceivedString,1,9)); // Pump status
				sPort.nCommStatus := STRING_TO_INT(mid(sPort.sLastReceivedString,1,10)); // Communication status
				//set next state
				sPort.nState := 4;
			ELSE
				sPort.nState := -3;  //place holder for action on failure
			END_IF
		4: //Received message should be <STX>Kx<CR>
			IF left(sPort.sLastReceivedString,2) = '$02K' THEN
				n := STRING_TO_INT(mid(sPort.sLastReceivedString,1,3));  //do nothing with this, just clear the flag
				//set next state
				sPort.nState := SEL(n = 0, 5, 6); //no keys pressed means can skip the key reset
			ELSE
				sPort.nState := -4;  //place holder for action on failure
			END_IF
		5: //No confirmation message expected after key clear
			sPort.nState := 6;  //go to speed request
		6: //Received message should be <STX>S+nnnn.n<CR>
			IF left(sPort.sLastReceivedString,2) = '$02S' THEN
				//sPort.bDirection := SEL((mid(sPort.sLastReceivedString,1,3) = '+'), FALSE, TRUE); //-/0 is reverse, +/1 is forward
				IF sPort.bRun THEN
					sPort.fSpeedPV := STRING_TO_LREAL(mid(sPort.sLastReceivedString,6,4));
				ELSE
					sPort.fSpeedPV := 0.0;
				END_IF				
				
				//set next state
				IF sPort.fSpeedSP_RQ >= 0.0  OR (sPort.nRun_RQ = 1) THEN //JRW issue #1 set speed every time pump is started to avoid pump running in wrong direction or wrong speed.
					sPort.nState := 7;
				ELSIF sPort.nRun_RQ <> -1 THEN
					sPort.nState := 8;
				ELSIF sPort.nLocal_RQ = 0 THEN
					sPort.nState := 10;
				ELSIF sPort.nLocal_RQ = 1 THEN
					sPort.nState := 11;
				ELSE
					sPort.nState := 3;
				END_IF
			ELSE
				sPort.nState := -6;  //place holder for action on failure
			END_IF
		7: //Received message should be <ACK>
			IF sPort.sLastReceivedString = '$06' THEN
				//set next state
				IF sPort.nRun_RQ <> -1 THEN
					sPort.nState := 8;
				ELSIF sPort.nLocal_RQ = 0 THEN
					sPort.nState := 10;
				ELSIF sPort.nLocal_RQ = 1 THEN
					sPort.nState := 11;
				ELSE
					sPort.nState := 3;
				END_IF
			ELSE
				sPort.nState := -7;  //place holder for action on failure
			END_IF
		8: //Received message should be <ACK>
			IF sPort.sLastReceivedString = '$06' THEN
				//set next state
				IF sPort.nLocal_RQ = 0 THEN
					sPort.nState := 10;
				ELSIF sPort.nLocal_RQ = 1 THEN
					sPort.nState := 11;
				ELSE
					sPort.nState := 3;
				END_IF
			ELSE
				sPort.nState := -8;  //place holder for action on failure
			END_IF
		10: //Received message should be <ACK><ACK>
			IF sPort.sLastReceivedString = '$06$06' THEN
				//set next state
				sPort.nState := 3;
			ELSE
				sPort.nState := -10;  //place holder for action on failure
			END_IF
		11: //Received message should be <ACK><ACK>
			IF sPort.sLastReceivedString = '$06$06' THEN
				//set next state
				sPort.nState := 3;
			ELSE
				sPort.nState := -11;  //place holder for action on failure
			END_IF
		END_CASE
	END_IF
	sPort.bListening := FALSE;
END_IF

END_FUNCTION_BLOCK

// ---- POUs/Wiesler/Masterflex/fbMasterflexSerial.TcPOU
FUNCTION_BLOCK fbMasterflexSerial
VAR
	// Comm buffers
	RxBufferMT			: ComBuffer;	// Receive data buffer for Mettler Toledo
	TxBufferMT			: ComBuffer;	// Transmit data buffer for Mettler Toledo
	// background communication with the EL6002 port
	fbPortCtrl		: SerialLineControl; // must be called every scan
	bPortCtrlError	: BOOL;
	ePortCtrlErrorID	: ComError_t;
	// Variables for sending data
	sSendString: STRING;
	fbSend		: SendString;
	bSendBusy	: BOOL;
	eSendErrorID: ComError_t;


	// Variables for receiving data
	fbReceive		: ReceiveString;
	sReceivedString	: STRING;
	bStringReceived	: BOOL;
	bReceiveBusy	: BOOL;
	bReceiveError	: BOOL;
	eReceiveErrorID	: ComError_t;
	
END_VAR

VAR_IN_OUT
	sPort : sMasterflexPort;
END_VAR

// *********************************************************************************
// The SerialLineControl function block is supposed to be called in every PLC cycle.
// It communicates with the serial line hardware device and transmits or receives data.
// The SerialLineControl can be called in the standard task (e.g.for PcCOM port usage) 
// or in a separate fast task (e.g.for terminal usage) as well.
// A fast separate task will be necessary at high baud rates or with KL6001 terminals 
// which have a small process image (3 or 5 data bytes only)
// **********************************************************************************

// background communication with the Port terminal
fbPortCtrl(
	Mode:= SERIALLINEMODE_EL6_22B, 
	pComIn:= ADR(sPort.stIn_Port), 
	pComOut:= ADR(sPort.stOut_Port), 
	SizeComIn:= UINT_TO_INT(SIZEOF(sPort.stIn_Port)), 
	Error=> , 
	ErrorID=> , 
	TxBuffer:= TxBufferMT, 
	RxBuffer:= RxBufferMT );
IF fbPortCtrl.Error THEN
	bPortCtrlError := TRUE;
	ePortCtrlErrorID := fbPortCtrl.ErrorID;
END_IF


// Call the send block if the sSendString has a value to send.
// Also call the block as long as it is busy to finish a transmission.
// When the transmission is complete clear sSendString to prepare for next string to send
IF len(sPort.sSendString) > 0 THEN
	fbSend(	SendString:= sPort.sSendString,
			TXbuffer:= TxBufferMT,
			Busy=> bSendBusy,
			Error=> );
	IF fbSend.Error <> COMERROR_NOERROR THEN
		eSendErrorID := fbSend.Error;
	END_IF
	IF NOT bSendBusy THEN
		sPort.sSendString := '';
	END_IF
END_IF

//	Receive string data:
//	The block receives any data strings ending with RxSuffix characters.	
fbReceive(
	Prefix:= '',
	Suffix:= sPort.sRxSuffix,
	Timeout:= T#1s,
	ReceivedString:= sReceivedString,
	RXbuffer:= RxBufferMT,
	StringReceived=> bStringReceived,
	Busy=> bReceiveBusy,
	Error=> ,
	RxTimeout=> sPort.bReceiveTimeout );
IF fbReceive.Error <> COMERROR_NOERROR THEN
	eReceiveErrorID := fbReceive.Error;
END_IF
IF bStringReceived THEN
	sPort.nReceiveCounter := sPort.nReceiveCounter + 1;
	sPort.sLastReceivedString := sReceivedString;
END_IF

END_FUNCTION_BLOCK

// ---- POUs/FlowCalibration/FlowCalSequence.TcPOU
FUNCTION_BLOCK FlowCalSequence
VAR_INPUT
	start : BOOL := FALSE;  //command to start
	setSpeedDuration : TIME := T#15S;  //Time to allow flow to stabilize before starting run
	runTestDuration : TIME := T#3M; //Time to collect liquid on the scale
	runTestWeight : LREAL := 20.0; // run for 100 grams minimum quantity of fluid on the scale for a completed flowrate
	autoAdvance : BOOL := TRUE; //Determines if the test should automatically start the next flowrate.  Sometimes the flow is too much and the collection vessel has to be emptied
	tubingType :INT := 14;
END_VAR
VAR_IN_OUT
	fq : FQ1; //flow totalizer
	pump : sMasterflexPort;
	FTOLS: OLSResult;
	pumpOLS: OLSResult;
END_VAR
VAR_OUTPUT
	startTimes : ARRAY[1..100] OF ULINT;
	endTimes : ARRAY[1..100] OF ULINT;
	flowTotal : ARRAY[1..100] OF LREAL;
	weight : ARRAY[1..100] OF LREAL;
	flowRate : ARRAY[1..100] OF LREAL;
	scaleRate : ARRAY[1..100] OF LREAL;
	calibrationStatus : UINT := 0;
END_VAR
VAR
	i : UINT := 0; // index
	n : UINT := 24;  //number of points to test
	t : LREAL := 0.0; //temporary variable
	tol : LREAL := 5.0;  //tolerance of the zeroing - weight must be below this to have successfully zero'd
	R2Tol : LREAL := 0.95; //tolerance of the OLS fit
	flowCalMTol : LREAL := 0.05; //tolerance for slope
	flowCalBTol : LREAL := 0.05; //tolerance for intercept
	OLSFlowTemp : OLSResult;
	OLSPumpTemp : OLSResult;
	sp : ARRAY [1..100] OF LREAL := [10.0, 20.0, 30.0, 40.0, 50.0, 60.0, 70.0, 80.0, 90.0, 100.0, 
                                    125.0, 150.0, 175.0, 200.0, 225.0, 250.0, 275.0, 300.0, 350.0, 400.0,
                                    450.0, 500.0, 550.0, 600.0, 0.0, 0.0, 0.0, 0.0, 0.0, 0.0,
                                    0.0, 0.0, 0.0, 0.0, 0.0, 0.0, 0.0, 0.0, 0.0, 0.0,
                                    0.0, 0.0, 0.0, 0.0, 0.0, 0.0, 0.0, 0.0, 0.0, 0.0,
                                    0.0, 0.0, 0.0, 0.0, 0.0, 0.0, 0.0, 0.0, 0.0, 0.0,
                                    0.0, 0.0, 0.0, 0.0, 0.0, 0.0, 0.0, 0.0, 0.0, 0.0,
                                    0.0, 0.0, 0.0, 0.0, 0.0, 0.0, 0.0, 0.0, 0.0, 0.0,
                                    0.0, 0.0, 0.0, 0.0, 0.0, 0.0, 0.0, 0.0, 0.0, 0.0,
                                    0.0, 0.0, 0.0, 0.0, 0.0, 0.0, 0.0, 0.0, 0.0, 0.0
									];

	setSpeed : SFCStepType;
	runTest : SFCStepType;
	recordTest : SFCStepType;
	calcCalibration : SFCStepType;
END_VAR

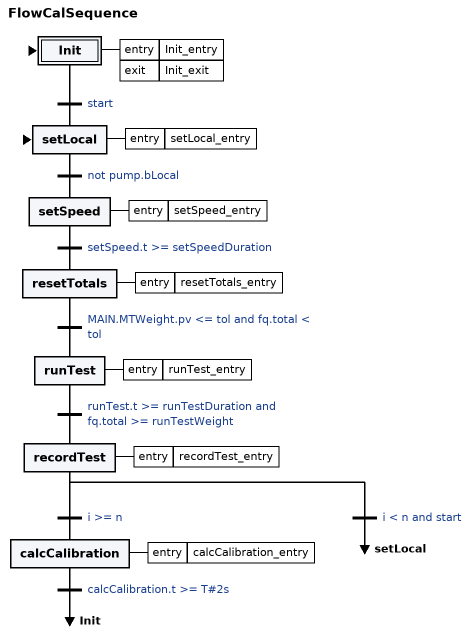
INITIAL_STEP Init:
    Init_entry(P1);  // entry action
    Init_exit(P0);  // exit action
END_STEP
TRANSITION FROM Init TO setLocal
    := start;
END_TRANSITION
STEP setLocal:
    setLocal_entry(P1);  // entry action
END_STEP
TRANSITION FROM setLocal TO setSpeed
    := not pump.bLocal;
END_TRANSITION
STEP setSpeed:
    setSpeed_entry(P1);  // entry action
END_STEP
TRANSITION FROM setSpeed TO resetTotals
    := setSpeed.t >= setSpeedDuration;
END_TRANSITION
STEP resetTotals:
    resetTotals_entry(P1);  // entry action
END_STEP
TRANSITION FROM resetTotals TO runTest
    := MAIN.MTWeight.pv <= tol and fq.total < tol;
END_TRANSITION
STEP runTest:
    runTest_entry(P1);  // entry action
END_STEP
TRANSITION FROM runTest TO recordTest
    := runTest.t >= runTestDuration and fq.total >= runTestWeight;
END_TRANSITION
STEP recordTest:
    recordTest_entry(P1);  // entry action
END_STEP
TRANSITION FROM recordTest TO calcCalibration
    := i >= n;
END_TRANSITION
STEP calcCalibration:
    calcCalibration_entry(P1);  // entry action
END_STEP
TRANSITION FROM recordTest TO setLocal
    := i < n and start;
END_TRANSITION
TRANSITION FROM calcCalibration TO Init
    := calcCalibration.t >= T#2s;
END_TRANSITION

ACTION resetTotals_entry:
fq.resetRQ := TRUE; //reset the totalizer
MAIN.MTSendString := 'ZI$0D$0A';  //Zero Immediately the scale
END_ACTION

ACTION Init_exit:
FOR i := 1 TO n DO
	startTimes[i] := 0;
	endTimes[i] := 0;
	flowTotal[i] := 0.0;
	weight[i] := 0.0;
	flowRate[i] := 0.0;	
	scaleRate[i] := 0.0;	
END_FOR
i := 0;
calibrationStatus := 2; //In process
END_ACTION

ACTION setSpeed_entry:
//Send speed setpoint
IF sp[i] > 0.1 THEN
	pump.nRun_RQ := 1; //start pump
	pump.fSpeedSP_RQ := sp[i];
ELSE
	pump.nRun_RQ := 0; //stop pump
	pump.fSpeedSP_RQ := 0.0;
END_IF
END_ACTION

ACTION runTest_entry:
MAIN.MTSendString := 'SIR$0D$0A'; //Send weight value Immediately and Repeat
startTimes[i] := unixTime;
END_ACTION

ACTION setLocal_entry:
i := i + 1;
IF pump.bLocal THEN
	pump.nLocal_RQ := 0;  //put pump in remote
END_IF
END_ACTION

ACTION Init_entry:
//reset for next calibration
start := FALSE;
END_ACTION

ACTION calcCalibration_entry:
//Stop pump
pump.nRun_RQ := 0; //stop pump

//run data analysis to determine new calibration values
//Check fit of flow data vs. scale data
OLSFlowTemp := ols(x := flowRate, y := scaleRate, length := n);
//Check fit of pump speed data vs. scale data
OLSPumpTemp := ols(x := scaleRate, y := sp, length := n);

//Determine maximum x value of flow data, this is just for the test of intercept
//Expect intercept to be 'near 0.0', so knowing the range of x values is
//necessary to determine what is 'close'
t := 0.0;
FOR i := 1 TO n DO
	t := MAX(t, flowRate[i]);	
END_FOR
IF t = 0.0 THEN //ensure no divide by zero
	t := 1.0;
END_IF

//Check Linearity, slope, and intercept (range and zero)
IF OLSFlowTemp.status <> 0 OR 							//OLS failed
		OLSFlowTemp.R2 < R2Tol OR 						//Not a good line fit
		ABS(1-OLSFlowTemp.m) > flowCalMTol OR  			//Slope not close to 1
		ABS(OLSFlowTemp.b/t) > flowCalBTol THEN			//Intercept is greater than tolerance % of scale
	calibrationStatus := 3; //Failed FT calibration
ELSE
	// Check for pump speed vs. flow 
	IF OLSFlowTemp.status <> 0 OR 						//OLS failed
			OLSFlowTemp.R2 < R2Tol THEN					//Not a good line fit
		calibrationStatus := 4; //Failed pump speed calibration
	ELSE
		calibrationStatus := 1; //Success
		//set both calibrations
		FTOLS := OLSFlowTemp;
		pumpOLS := OLSPumpTemp;  //All checks were good, the calibration is successful.
	END_IF
END_IF
END_ACTION

ACTION recordTest_entry:
endTimes[i] := unixTime;
flowTotal[i] := fq.total;
weight[i] := MAIN.MTWeight.pv;
t := ULINT_TO_LREAL(endTimes[i] - startTimes[i])/1000.0/60.0; //Test duration in minutes
flowRate[i] := flowTotal[i]/t;
scaleRate[i] := weight[i]/t;
IF NOT autoAdvance THEN
	start := FALSE;
END_IF
END_ACTION

END_FUNCTION_BLOCK

// ---- POUs/FlowCalibration/OLS.TcPOU
FUNCTION OLS : OLSResult
VAR_INPUT
	x : ARRAY [1..100] OF LREAL;
	y : ARRAY [1..100] OF LREAL;
	length : UINT;
END_VAR
VAR
	fLength: LREAL;
	f : LREAL;
	i : UINT := 0;
	xSquaredSum : LREAL := 0;
	xySum : LREAL := 0;
	xBar : LREAL := 0;
	yBar : LREAL := 0;
	xSum : LREAL := 0;
	ySum : LREAL := 0;
	
	fx : LREAL := 0; // y = fx = m * x + b
	SSE : LREAL := 0; // sum of square error
	SST : LREAL := 0; // sum of squares total

END_VAR

IF length < 2 OR length > 100 THEN
	OLS.status := 1;
	RETURN;
END_IF

fLength := UINT_TO_LREAL(length);

FOR i := 1 TO length DO
	xSquaredSum := xSquaredSum + x[i] * x[i];
	xySum := xySum + x[i] * y[i];
	xSum := xSum + x[i];
	ySum := ySum + y[i];
END_FOR

xBar := xSum / fLength;
yBar := ySum / fLength;

f := xSquaredSum - (fLength * xBar * xBar);
IF ABS(f) < 0.001 THEN // TODO: determine proper tolerance
	OLS.status := 2;
	RETURN;
END_IF

OLS.m := (xySum - (fLength * xBar * yBar)) / f;
OLS.b := yBar - (OLS.m * xBar);

FOR i := 1 TO length DO
	fx := OLS.m * x[i] + OLS.b;
	SSE := SSE + ((y[i] - fx) * (y[i] - fx));
	SST := SST + ((y[i] - yBar) * (y[i] - yBar));
END_FOR

OLS.R2 := 1 - SSE / SST;

END_FUNCTION

// ---- POUs/Wiesler/AI1.TcPOU
FUNCTION_BLOCK AI1
VAR_IN_OUT
	ai : AI;
END_VAR
VAR_OUTPUT
END_VAR
VAR
END_VAR

IF ai.sim.simEnable THEN
	ai.pv := ai.sim.simValue;
ELSE
	ai.pv := ai.scale.euLo + (ai.raw - ai.scale.rawLo)*(ai.scale.euHi - ai.scale.euLo)/(ai.scale.rawHi - ai.scale.rawLo);
	IF ai.loCutEnable AND ai.pv < ai.loCut THEN
		ai.pv := 0.0;
	END_IF
END_IF

END_FUNCTION_BLOCK

// ---- POUs/Wiesler/fbMovingAverage.TcPOU
FUNCTION_BLOCK fbMovingAverage
VAR CONSTANT
	arrSize : UINT := 3000; //Do not change online.
END_VAR
VAR_INPUT
	in : LREAL;
	size : UINT := 1000;
END_VAR
VAR_OUTPUT
	out : LREAL;
END_VAR
VAR
	wkSize : UINT;
	start : UINT := arrSize - 1;
	vals : ARRAY[0..arrSize - 1] OF LREAL := [arrSize(0.0)];
	lastSize : UINT := 0;
	end : UINT;
	i : UINT;
END_VAR
VAR_IN_OUT
END_VAR

wkSize := LIMIT(1, size, arrSize); //make sure size is in limits
start := (start + 1) MOD arrSize;
IF lastSize <> wkSize THEN //moving average size has changed, need to totally recalculate out
	vals[start] := in;
	out := 0.0;
	FOR i := 1 TO size DO
		out := out + vals[(start + 1 + arrSize - i) MOD arrSize];
	END_FOR
	out := out/UINT_TO_LREAL(size);
	lastSize := wkSize;
ELSE
	out := out + (in - vals[(start + arrSize - size) MOD arrSize])/UINT_TO_LREAL(size);
	vals[start] := in;
END_IF

END_FUNCTION_BLOCK

// ---- POUs/Wiesler/Datalog/fbDatalogger_100ms.TcPOU
FUNCTION_BLOCK fbDatalogger_100ms

VAR CONSTANT
	nRate : DINT := 100;
	nPoints : DINT := 1000 / nRate;
END_VAR

VAR_INPUT
	fData : LREAL;
END_VAR
VAR_OUTPUT
	afLog : ARRAY[0..(nPoints-1)] OF LREAL;
	nLogJSTime : ULINT := 0;
END_VAR
VAR
	afCache : ARRAY[0..(nPoints-1)] OF LREAL;
	nCount : DINT := 0;
END_VAR

IF unixTime MOD DINT_TO_ULINT(nRate) = 0 THEN
	// Fill up the SampleArray
	afCache[nCount] := fData;
	// Increase the sampleIndex
	nCount := nCount + 1;
END_IF

IF nCount >= nPoints THEN
	// Copy values into log array
	afLog := afCache;
	// Increment log index to tell watching external logger the data has changed
	nLogJSTime := unixTime;
	// Reset count
	nCount := 0;
END_IF

END_FUNCTION_BLOCK

// ---- POUs/Wiesler/Datalog/fbDatalogger_1ms.TcPOU
FUNCTION_BLOCK fbDatalogger_1ms

VAR CONSTANT
	nRate : DINT := 1;
	nPoints : DINT := 1000 / nRate;
END_VAR

VAR_INPUT
	fData : LREAL;
END_VAR
VAR_OUTPUT
	afLog : ARRAY[0..(nPoints-1)] OF LREAL;
	nLogJSTime : ULINT := 0;
END_VAR
VAR
	afCache : ARRAY[0..(nPoints-1)] OF LREAL;
	nCount : DINT := 0;
END_VAR

IF unixTime MOD DINT_TO_ULINT(nRate) = 0 THEN
	// Fill up the SampleArray
	afCache[nCount] := fData;
	// Increase the sampleIndex
	nCount := nCount + 1;
END_IF

IF nCount >= nPoints THEN
	// Copy values into log array
	afLog := afCache;
	// Increment log index to tell watching external logger the data has changed
	nLogJSTime := unixTime;
	// Reset count
	nCount := 0;
END_IF

END_FUNCTION_BLOCK

// ---- POUs/Wiesler/Datalog/fbDatalogger_10ms.TcPOU
FUNCTION_BLOCK fbDatalogger_10ms

VAR CONSTANT
	nRate : DINT := 10;
	nPoints : DINT := 1000 / nRate;
END_VAR

VAR_INPUT
	fData : LREAL;
END_VAR
VAR_OUTPUT
	afLog : ARRAY[0..(nPoints-1)] OF LREAL;
	nLogJSTime : ULINT := 0;
END_VAR
VAR
	afCache : ARRAY[0..(nPoints-1)] OF LREAL;
	nCount : DINT := 0;
END_VAR

IF unixTime MOD DINT_TO_ULINT(nRate) = 0 THEN
	// Fill up the SampleArray
	afCache[nCount] := fData;
	// Increase the sampleIndex
	nCount := nCount + 1;
END_IF

IF nCount >= nPoints THEN
	// Copy values into log array
	afLog := afCache;
	// Increment log index to tell watching external logger the data has changed
	nLogJSTime := unixTime;
	// Reset count
	nCount := 0;
END_IF

END_FUNCTION_BLOCK

// ---- POUs/MTSerial.TcPOU
PROGRAM MTSerial
VAR
	// Comm buffers
	RxBufferMT			: ComBuffer;	// Receive data buffer for Mettler Toledo
	TxBufferMT			: ComBuffer;	// Transmit data buffer for Mettler Toledo
	// background communication with the EL6002 port
	fbPortCtrl		: SerialLineControl; // must be called every scan
	bPortCtrlError	: BOOL;
	ePortCtrlErrorID	: ComError_t;
	// I/O variables for a EL6001 terminal
	stIn_Port AT %I*	: EL6inData22B;	// linked to the EL6002 in the TwinCAT System Manager
	stOut_Port AT %Q*	: EL6outData22B; // linked to the EL6002 in the TwinCAT System Manager
	
	// Variables for sending data
	fbSend		: SendString;
	bSendBusy	: BOOL;
	eSendErrorID: ComError_t;

	// Variables for receiving data
	fbReceive		: ReceiveString;
	sReceivedString	: STRING;
	bStringReceived	: BOOL;
	bReceiveBusy	: BOOL;
	bReceiveError	: BOOL;
	eReceiveErrorID	: ComError_t;
	bReceiveTimeout	: BOOL;
	nReceiveCounter	: UDINT := 0;
	sLastReceivedString: STRING;
END_VAR

VAR_IN_OUT
	sSendString: STRING;
	weight: sWeight;
END_VAR

// *********************************************************************************
// The SerialLineControl function block is supposed to be called in every PLC cycle.
// It communicates with the serial line hardware device and transmits or receives data.
// The SerialLineControl can be called in the standard task (e.g.for PcCOM port usage) 
// or in a separate fast task (e.g.for terminal usage) as well.
// A fast separate task will be necessary at high baud rates or with KL6001 terminals 
// which have a small process image (3 or 5 data bytes only)
// **********************************************************************************

// background communication with the Port terminal
fbPortCtrl(
	Mode:= SERIALLINEMODE_EL6_22B, 
	pComIn:= ADR(stIn_Port), 
	pComOut:= ADR(stOut_Port), 
	SizeComIn:= UINT_TO_INT(SIZEOF(stIn_Port)), 
	Error=> , 
	ErrorID=> , 
	TxBuffer:= TxBufferMT, 
	RxBuffer:= RxBufferMT );
IF fbPortCtrl.Error THEN
	bPortCtrlError := TRUE;
	ePortCtrlErrorID := fbPortCtrl.ErrorID;
END_IF


// Call the send block if the sSendString has a value to send.
// Also call the block as long as it is busy to finish a transmission.
// When the transmission is complete clear sSendString to prepare for next string to send
IF len(sSendString) > 0 THEN
	fbSend(	SendString:= sSendString,
			TXbuffer:= TxBufferMT,
			Busy=> bSendBusy,
			Error=> );
	IF fbSend.Error <> COMERROR_NOERROR THEN
		eSendErrorID := fbSend.Error;
	END_IF
	IF NOT bSendBusy THEN
		sSendString := '';
	END_IF
END_IF

//	Receive string data:
//	The block receives any data strings ending with an CRLF characters.	
fbReceive(
	Prefix:= '',
	Suffix:= '$0D$0A',
	Timeout:= T#1s,
	ReceivedString:= sReceivedString,
	RXbuffer:= RxBufferMT,
	StringReceived=> bStringReceived,
	Busy=> bReceiveBusy,
	Error=> ,
	RxTimeout=> bReceiveTimeout );
IF fbReceive.Error <> COMERROR_NOERROR THEN
	eReceiveErrorID := fbReceive.Error;
END_IF
IF bStringReceived THEN
	nReceiveCounter := nReceiveCounter + 1;
	sLastReceivedString := sReceivedString;
	weight := MT_SICS_TO_Weight(weight, sLastReceivedString);
END_IF

END_PROGRAM

// ---- POUs/Wiesler/MT_SICS_TO_Weight.TcPOU
FUNCTION MT_SICS_TO_Weight : sWeight
VAR_INPUT
	lastWeight: sWeight;
	MT_SICS_Message: STRING;
END_VAR
VAR
	response: STRING;
END_VAR

MT_SICS_TO_Weight.pv := lastWeight.pv;
MT_SICS_TO_Weight.status := lastWeight.status;

IF mid(MT_SICS_Message, 2, 1) = 'S ' THEN
	IF mid(MT_SICS_Message, 1, 3) = 'S' THEN
		MT_SICS_TO_Weight.status := 'Stable';
	ELSE
		MT_SICS_TO_Weight.status := 'Dynamic';
	END_IF
	MT_SICS_TO_Weight.pv := STRING_TO_LREAL(mid(MT_SICS_Message, 10, 5));
END_IF

END_FUNCTION

// ---- POUs/FlowCheck.TcPOU
PROGRAM FlowCheck
VAR_INPUT
	start : BOOL := FALSE;
	setSpeedDuration : TIME := T#15S;
	runTestDuration : TIME := T#15S;
	runTestWeight : lreal := 10.0; // run for 100 grams
	autoAdvance : BOOL := TRUE;
END_VAR
VAR_OUTPUT
	startTimes : ARRAY[1..50] OF ULINT;
	endTimes : ARRAY[1..50] OF ULINT;
	FQA : ARRAY[1..50] OF LREAL;
	FQB : ARRAY[1..50] OF LREAL;
	FQC : ARRAY[1..50] OF LREAL;
	weight : ARRAY[1..50] OF LREAL;
	FTA_mean : ARRAY[1..50] OF LREAL;
	FTB_mean : ARRAY[1..50] OF LREAL;
	FTC_mean : ARRAY[1..50] OF LREAL;
	P9999Atubing : ARRAY[1..50] OF INT;
	P9999Btubing : ARRAY[1..50] OF INT;
END_VAR
VAR
	i : UINT := 0; // index
	n : UINT := 25;
	t : LREAL := 0.0;
	tol : LREAL := 5.0;
	//spA : ARRAY [1..50] OF LREAL := [10.0, 20.0, 30.0, 40.0, 50.0, 60.0, 70.0, 80.0, 90.0, 100.0, 
    //                                125.0, 150.0, 175.0, 200.0, 225.0, 250.0, 275.0, 300.0,
    //                                350.0, 400.0, 450.0, 500.0, 550.0, 600.0,
	//								0.0,0.0,0.0,0.0,0.0,0.0,0.0,0.0,0.0,0.0,0.0,0.0,0.0,0.0,0.0,0.0,0.0,0.0,0.0,0.0,0.0,0.0,0.0,0.0];
	spA : ARRAY [1..50] OF LREAL := [10.0, 20.0, 30.0, 40.0, 50.0, 60.0, 70.0, 80.0, 90.0, 100.0, 
                                    110.0, 120.0, 130.0, 140.0, 150.0, 0.0, 0.0, 0.0,
                                    0.0, 0.0, 0.0, 0.0, 0.0, 0.0,
									0.0,0.0,0.0,0.0,0.0,0.0,0.0,0.0,0.0,0.0,0.0,0.0,0.0,0.0,0.0,0.0,0.0,0.0,0.0,0.0,0.0,0.0,0.0,0.0];
	spB : ARRAY [1..50] OF LREAL := [0.0,0.0,0.0,0.0,0.0,0.0,0.0,0.0,0.0,0.0,0.0,0.0,0.0,0.0,0.0,0.0,0.0,0.0,0.0,0.0,0.0,0.0,0.0,0.0,
									0.0,0.0,0.0,0.0,0.0,0.0,0.0,0.0,0.0,0.0,0.0,0.0,0.0,0.0,0.0,0.0,0.0,0.0,0.0,0.0,0.0,0.0,0.0,0.0
	];
	//								0.0, 20.0, 30.0, 40.0, 50.0, 60.0, 70.0, 80.0, 90.0, 100.0, 
    //                                125.0, 150.0, 175.0, 200.0, 225.0, 250.0, 275.0, 300.0,
    //                                350.0, 400.0, 450.0, 500.0, 550.0, 600.0];
	//spA : ARRAY [1..50] OF LREAL := [0.0,0.0,0.0,0.0,0.0,0.0,0.0,0.0,0.0,0.0,0.0,0.0,0.0,0.0,0.0,0.0,0.0,0.0,0.0,0.0,0.0,0.0,0.0,0.0,
	//								0.0, 20.0, 30.0, 40.0, 50.0, 60.0, 70.0, 80.0, 90.0, 100.0, 
    //                                125.0, 150.0, 175.0, 200.0, 225.0, 250.0, 275.0, 300.0,
    //                                350.0, 400.0, 450.0, 500.0, 550.0, 600.0];
	//sp : ARRAY [1..50] OF LREAL := [51.0, 58.0, 64.0, 79.0, 97.0, 112.0, 128.0, 151.0, 210.0, 280.0, 335.0, 410.0, 480.0, 600.0];
	//sp : ARRAY [1..50] OF LREAL := [335.0, 410.0, 480.0, 600.0];
	setSpeed : SFCStepType;
	runTest : SFCStepType;
	recordTest : SFCStepType;
END_VAR

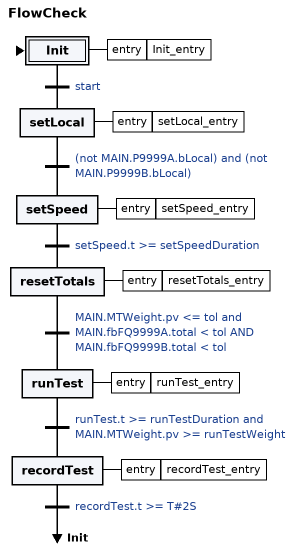
INITIAL_STEP Init:
    Init_entry(P1);  // entry action
END_STEP
TRANSITION FROM Init TO setLocal
    := start;
END_TRANSITION
STEP setLocal:
    setLocal_entry(P1);  // entry action
END_STEP
TRANSITION FROM setLocal TO setSpeed
    := (not MAIN.P9999A.bLocal) and (not MAIN.P9999B.bLocal);
END_TRANSITION
STEP setSpeed:
    setSpeed_entry(P1);  // entry action
END_STEP
TRANSITION FROM setSpeed TO resetTotals
    := setSpeed.t >= setSpeedDuration;
END_TRANSITION
STEP resetTotals:
    resetTotals_entry(P1);  // entry action
END_STEP
TRANSITION FROM resetTotals TO runTest
    := MAIN.MTWeight.pv <= tol and MAIN.fbFQ9999A.total < tol AND MAIN.fbFQ9999B.total < tol;
END_TRANSITION
STEP runTest:
    runTest_entry(P1);  // entry action
END_STEP
TRANSITION FROM runTest TO recordTest
    := runTest.t >= runTestDuration and MAIN.MTWeight.pv >= runTestWeight;
END_TRANSITION
STEP recordTest:
    recordTest_entry(P1);  // entry action
END_STEP
TRANSITION FROM recordTest TO Init
    := recordTest.t >= T#2S;
END_TRANSITION

ACTION Init_entry:
IF i >= n THEN
	MAIN.P9999A.nRun_RQ := 0; //stop pump
	MAIN.P9999B.nRun_RQ := 0; //stop pump
	start := FALSE;
	i := 0;
END_IF
MAIN.logActive := FALSE;
END_ACTION

ACTION resetTotals_entry:
MAIN.fbFQ9999A.resetRQ := TRUE;
MAIN.fbFQ9999B.resetRQ := TRUE;
MAIN.fbFQ9999C.resetRQ := TRUE;
MAIN.MTSendString := 'ZI$0D$0A';
MAIN.logActive := TRUE;
END_ACTION

ACTION setSpeed_entry:
i := i + 1;
startTimes[i] := 0;
endTimes[i] := 0;
FQA[i] := 0;
FQB[i] := 0;
FQC[i] := 0;
weight[i] := 0;
FTA_mean[i] := 0;
FTB_mean[i] := 0;
FTC_mean[i] := 0;
IF spA[i] > 0.1 THEN
	MAIN.P9999A.nRun_RQ := 1; //start pump
	MAIN.P9999A.fSpeedSP_RQ := spA[i];
ELSE
	MAIN.P9999A.nRun_RQ := 0; //stop pump
	MAIN.P9999A.fSpeedSP_RQ := 0.0;
END_IF
	
IF spB[i] > 0.1 THEN
	MAIN.P9999B.nRun_RQ := 1; //start pump
	MAIN.P9999B.fSpeedSP_RQ := spB[i];
ELSE
	MAIN.P9999B.nRun_RQ := 0; //stop pump
	MAIN.P9999B.fSpeedSP_RQ := 0.0;
END_IF

P9999Atubing[i] := MAIN.P9999A.nTubeSize;
P9999Btubing[i] := MAIN.P9999B.nTubeSize;
END_ACTION

ACTION setLocal_entry:
IF MAIN.P9999A.bLocal THEN
	MAIN.P9999A.nLocal_RQ := 0;  //put pump in remote
END_IF
IF MAIN.P9999B.bLocal THEN
	MAIN.P9999B.nLocal_RQ := 0;  //put pump in remote
END_IF
END_ACTION

ACTION recordTest_entry:
endTimes[i] := unixTime;
FQA[i] := MAIN.fbFQ9999A.total;
FQB[i] := MAIN.fbFQ9999B.total;
FQC[i] := MAIN.fbFQ9999C.total;
weight[i] := MAIN.MTWeight.pv;
t := DWORD_TO_LREAL(TIME_TO_DWORD(runTestDuration))/1000.0/60.0;
FTA_mean[i] := MAIN.fbFQ9999A.total/t;
FTB_mean[i] := MAIN.fbFQ9999B.total/t;
FTC_mean[i] := MAIN.fbFQ9999C.total/t;
IF NOT autoAdvance THEN
	start := FALSE;
END_IF
END_ACTION

ACTION runTest_entry:
MAIN.MTSendString := 'SIR$0D$0A';
startTimes[i] := unixTime;
END_ACTION

END_PROGRAM

// ---- POUs/Wiesler/FlowConcentrationControl/StartStopSequence_CC1Test.TcPOU
PROGRAM StartStopSequence_CC1Test
VAR_INPUT
	start : BOOL := FALSE;
	setSpeedDuration : TIME := T#0S;
	autoAdvance : BOOL := TRUE;
END_VAR
VAR_OUTPUT
	startTimes : ARRAY[1..50] OF ULINT;
	endTimes : ARRAY[1..50] OF ULINT;

	P9999Atubing : ARRAY[1..50] OF INT;
	P9999Btubing : ARRAY[1..50] OF INT;
END_VAR
VAR
	i : UINT := 0; // index
	n : UINT := 25;
	t : LREAL := 0.0;
	tol : LREAL := 5.0;
	spTotal : ARRAY [1..50] OF LREAL := [100.0,100.0,100.0,0.0,0.0,0.0,0.0,0.0,0.0,0.0,0.0,0.0,0.0,0.0,0.0,0.0,0.0,0.0,0.0,0.0,0.0,0.0,0.0,0.0, 0.0,
									0.0,0.0,0.0,0.0,0.0,0.0,0.0,0.0,0.0,0.0,0.0,0.0,0.0,0.0,0.0,0.0,0.0,0.0,0.0,0.0,0.0,0.0,0.0,0.0,0.0];
	//spTotal : ARRAY [1..50] OF LREAL := [100.0, 150.0, 200.0, 300.0, 150.0, 100.0, 80.0, 80.0, 90.0, 100.0, 
    //                                110.0, 120.0, 130.0, 140.0, 150.0, 0.0, 0.0, 0.0,
    //                                0.0, 0.0, 0.0, 0.0, 0.0, 0.0,
	//								0.0,0.0,0.0,0.0,0.0,0.0,0.0,0.0,0.0,0.0,0.0,0.0,0.0,0.0,0.0,0.0,0.0,0.0,0.0,0.0,0.0,0.0,0.0,0.0];
	spConc : ARRAY [1..50] OF LREAL := [1.0, 1.0, 1.0, 1.0, 1.0, 1.0, 1.0, 1.0, 1.0, 1.0, 
                                    1.0, 1.0, 1.0, 1.0, 1.0, 0.0, 0.0, 0.0,
                                    0.0, 0.0, 0.0, 0.0, 0.0, 0.0,
									0.0,0.0,0.0,0.0,0.0,0.0,0.0,0.0,0.0,0.0,0.0,0.0,0.0,0.0,0.0,0.0,0.0,0.0,0.0,0.0,0.0,0.0,0.0,0.0];
	stopTime : ARRAY [1..50] OF TIME := [T#0.5M, T#0.5M, T#0.5M, T#10.0M, T#15.0M, T#30.0M, T#60.0M, T#120.0M, T#1.0M, T#1.0M, 
                                    T#1.0M, T#1.0M, T#1.0M, T#1.0M, T#1.0M, T#0.0M, T#0.0M, T#0.0M,
                                    T#0.0M, T#0.0M, T#0.0M, T#0.0M, T#0.0M, T#0.0M,
									T#0.0M,T#0.0M,T#0.0M,T#0.0M,T#0.0M,T#0.0M,T#0.0M,T#0.0M,T#0.0M,T#0.0M,T#0.0M,T#0.0M,T#0.0M,
									T#0.0M,T#0.0M,T#0.0M,T#0.0M,T#0.0M,T#0.0M,T#0.0M,T#0.0M,T#0.0M,T#0.0M,T#0.0M];
	runTime : ARRAY [1..50] OF TIME := [T#0.1M, T#0.1M, T#0.1M, T#1.0M, T#1.0M, T#1.0M, T#1.0M, T#1.0M, T#1.0M, T#1.0M, 
                                    T#1.0M, T#1.0M, T#1.0M, T#1.0M, T#1.0M, T#0.0M, T#0.0M, T#0.0M,
                                    T#0.0M, T#0.0M, T#0.0M, T#0.0M, T#0.0M, T#0.0M,
									T#0.0M,T#0.0M,T#0.0M,T#0.0M,T#0.0M,T#0.0M,T#0.0M,T#0.0M,T#0.0M,T#0.0M,T#0.0M,T#0.0M,T#0.0M,
									T#0.0M,T#0.0M,T#0.0M,T#0.0M,T#0.0M,T#0.0M,T#0.0M,T#0.0M,T#0.0M,T#0.0M,T#0.0M];
	
	setSpeed : SFCStepType;
	runTest : SFCStepType;
	recordTest : SFCStepType;
END_VAR

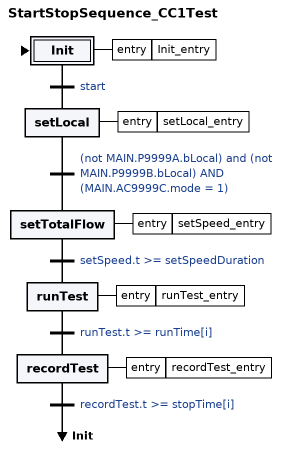
INITIAL_STEP Init:
    Init_entry(P1);  // entry action
END_STEP
TRANSITION FROM Init TO setLocal
    := start;
END_TRANSITION
STEP setLocal:
    setLocal_entry(P1);  // entry action
END_STEP
TRANSITION FROM setLocal TO setTotalFlow
    := (not MAIN.P9999A.bLocal) and (not MAIN.P9999B.bLocal) AND (MAIN.AC9999C.mode = 1);
END_TRANSITION
STEP setTotalFlow:
    setSpeed_entry(P1);  // entry action
END_STEP
TRANSITION FROM setTotalFlow TO runTest
    := setSpeed.t >= setSpeedDuration;
END_TRANSITION
STEP runTest:
    runTest_entry(P1);  // entry action
END_STEP
TRANSITION FROM runTest TO recordTest
    := runTest.t >= runTime[i];
END_TRANSITION
STEP recordTest:
    recordTest_entry(P1);  // entry action
END_STEP
TRANSITION FROM recordTest TO Init
    := recordTest.t >= stopTime[i];
END_TRANSITION

ACTION recordTest_entry:
endTimes[i] := unixTime;
MAIN.AC9999C.c.rq := 0; // set flow to 0 to stop pumps
t := DWORD_TO_LREAL(TIME_TO_DWORD(runTime[i]))/1000.0/60.0;

IF NOT autoAdvance THEN
	start := FALSE;
END_IF
END_ACTION

ACTION runTest_entry:
MAIN.MTSendString := 'SIR$0D$0A';
startTimes[i] := unixTime;
END_ACTION

ACTION resetTotals_entry:
MAIN.fbFQ9999A.resetRQ := TRUE;
MAIN.fbFQ9999B.resetRQ := TRUE;
MAIN.fbFQ9999C.resetRQ := TRUE;
MAIN.MTSendString := 'ZI$0D$0A';
MAIN.logActive := TRUE;
END_ACTION

ACTION setLocal_entry:
IF MAIN.P9999A.bLocal THEN
	MAIN.P9999A.nLocal_RQ := 0;  //put pump in remote
END_IF
IF MAIN.P9999B.bLocal THEN
	MAIN.P9999B.nLocal_RQ := 0;  //put pump in remote
END_IF

IF MAIN.AC9999C.mode <> 1 THEN 
	MAIN.AC9999C.mode := 1; // concentration control in auto
	MAIN.AC9999C.c.rq := 0; // set initial total flow
	MAIN.AC9999C.conc.rq := 1.0; // set initial concentration
	
END_IF
END_ACTION

ACTION setSpeed_entry:
i := i + 1;
startTimes[i] := 0;
endTimes[i] := 0;

MAIN.AC9999C.c.rq := spTotal[i];
MAIN.AC9999C.conc.rq := spConc[i];

P9999Atubing[i] := MAIN.P9999A.nTubeSize;
P9999Btubing[i] := MAIN.P9999B.nTubeSize;
END_ACTION

ACTION Init_entry:
IF i >= n THEN
	MAIN.AC9999C.mode := 0; // concentration control in manual
	MAIN.P9999A.nRun_RQ := 0; //stop pump
	MAIN.P9999B.nRun_RQ := 0; //stop pump
	start := FALSE;
	i := 0;
END_IF
MAIN.logActive := FALSE;
END_ACTION

END_PROGRAM

// ---- POUs/FlowCalibration/testOLS.TcPOU
FUNCTION_BLOCK testOLS
VAR_INPUT
END_VAR
VAR_OUTPUT
	result : INT := 0;
END_VAR
VAR
	OLSOut : OLSResult;
	y1 : ARRAY [1..100] OF LREAL := [  0.12548111,   2.48964043,   3.8531352 ,   5.02534211,
         6.19021734,   7.34772823,   8.5165989 ,   9.69657362,
        10.88234988,  12.06983084,  15.09756653,  18.07902939,
        21.10340477,  23.99898836,  26.91563451,  29.92832035,
        33.03966693,  35.97102658,  41.68383358,  46.98476969,
        53.01302749,  57.72483702,  63.22571341,  68.34296168, 0, 0, 0, 0, 0, 0,
		0, 0, 0, 0, 0, 0, 0, 0, 0, 0, 
		0, 0, 0, 0, 0, 0, 0, 0, 0, 0, 
		0, 0, 0, 0, 0, 0, 0, 0, 0, 0, 
		0, 0, 0, 0, 0, 0, 0, 0, 0, 0, 
		0, 0, 0, 0, 0, 0, 0, 0, 0, 0, 
		0, 0, 0, 0, 0, 0, 0, 0, 0, 0, 
		0, 0, 0, 0, 0, 0, 0, 0, 0, 0];
	x1 : ARRAY [1..100] OF LREAL := [ 10,  20,  30,  40,  50,  60,  70,  80,  90, 100, 125, 150, 175,
       200, 225, 250, 275, 300, 350, 400, 450, 500, 550, 600, 0, 0, 0, 0, 0, 0,
		0, 0, 0, 0, 0, 0, 0, 0, 0, 0, 
		0, 0, 0, 0, 0, 0, 0, 0, 0, 0, 
		0, 0, 0, 0, 0, 0, 0, 0, 0, 0, 
		0, 0, 0, 0, 0, 0, 0, 0, 0, 0, 
		0, 0, 0, 0, 0, 0, 0, 0, 0, 0, 
		0, 0, 0, 0, 0, 0, 0, 0, 0, 0, 
		0, 0, 0, 0, 0, 0, 0, 0, 0, 0];
	x2 : ARRAY [1..100] OF LREAL := [ 10,  10,  10,  10,  10,  10,  10,  10,  10, 10, 10, 10, 10,
       10, 10, 10, 10, 10, 10, 10, 10, 10, 10, 10, 0, 0, 0, 0, 0, 0,
		0, 0, 0, 0, 0, 0, 0, 0, 0, 0, 
		0, 0, 0, 0, 0, 0, 0, 0, 0, 0, 
		0, 0, 0, 0, 0, 0, 0, 0, 0, 0, 
		0, 0, 0, 0, 0, 0, 0, 0, 0, 0, 
		0, 0, 0, 0, 0, 0, 0, 0, 0, 0, 
		0, 0, 0, 0, 0, 0, 0, 0, 0, 0, 
		0, 0, 0, 0, 0, 0, 0, 0, 0, 0];
	n : INT; // length of data array
END_VAR

// testing if length is out of range
OLSOut := OLS(x:=x1, y:=y1, length:=1);
IF OLSOut.status <> 1 THEN
	result := result + 1;
END_IF

// testing if length is out of range
OLSOut := OLS(x:=x1, y:=y1, length:=101);
IF OLSOut.status <> 1 THEN
	result := result + 1;
END_IF

// testing if OLS results (m, b, R2) as expected
n := 24;
OLSOut := OLS(x:=x1, y:=y1, length:=n);
IF OLSOut.status <> 0 THEN
	result := result + 1;
	ELSE IF ABS(OLSOut.b - 0.554765) > 0.01 OR 
            ABS(OLSOut.m - 0.115292) > 0.01 OR
            ABS(OLSOut.R2 - 0.999126) > 0.01 THEN
		result := result + 1;
		END_IF
END_IF

OLSOut := OLS(x:=x2, y:=y1, length:=n);
IF OLSOut.status <> 2 THEN
	result := result + 1;
END_IF

END_FUNCTION_BLOCK

// ---- POUs/sonotecCalibration.TcPOU
PROGRAM sonotecCalibration
VAR_INPUT
	start : BOOL := FALSE;
	pumpA : BOOL := TRUE;
	setSpeedDuration : TIME := T#2M;
	runTestDuration : TIME := T#5M;
END_VAR
VAR_OUTPUT
	results : ARRAY[1..50] OF testResults;
END_VAR
VAR
	i : UINT := 0; // index
	n : UINT := 7;
	t : LREAL := 0.0;
	sp : ARRAY [1..50] OF LREAL := [80.0, 160.0, 240.0, 320.0, 400.0, 480.0, 560.0];
	//sp : ARRAY [1..50] OF LREAL := [51.0, 58.0, 64.0, 79.0, 97.0, 112.0, 128.0, 151.0, 210.0, 280.0, 335.0, 410.0, 480.0, 600.0];
	//sp : ARRAY [1..50] OF LREAL := [335.0, 410.0, 480.0, 600.0];
	setSpeed : SFCStepType;
	runTest : SFCStepType;
	recordTest : SFCStepType;
END_VAR

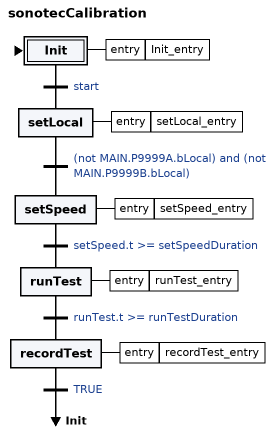
INITIAL_STEP Init:
    Init_entry(P1);  // entry action
END_STEP
TRANSITION FROM Init TO setLocal
    := start;
END_TRANSITION
STEP setLocal:
    setLocal_entry(P1);  // entry action
END_STEP
TRANSITION FROM setLocal TO setSpeed
    := (not MAIN.P9999A.bLocal) and (not MAIN.P9999B.bLocal);
END_TRANSITION
STEP setSpeed:
    setSpeed_entry(P1);  // entry action
END_STEP
TRANSITION FROM setSpeed TO runTest
    := setSpeed.t >= setSpeedDuration;
END_TRANSITION
STEP runTest:
    runTest_entry(P1);  // entry action
END_STEP
TRANSITION FROM runTest TO recordTest
    := runTest.t >= runTestDuration;
END_TRANSITION
STEP recordTest:
    recordTest_entry(P1);  // entry action
END_STEP
TRANSITION FROM recordTest TO Init
    := TRUE;
END_TRANSITION

ACTION setLocal_entry:
IF MAIN.P9999A.bLocal THEN
	MAIN.P9999A.nLocal_RQ := 0;  //put pump in remote
END_IF
IF MAIN.P9999B.bLocal THEN
	MAIN.P9999B.nLocal_RQ := 0;  //put pump in remote
END_IF
END_ACTION

ACTION runTest_entry:
MAIN.fbFQ9999A.resetRQ := TRUE;
MAIN.fbFQ9999B.resetRQ := TRUE;
MAIN.fbFQ9999C.resetRQ := TRUE;
END_ACTION

ACTION setSpeed_entry:
i := i + 1;
results[i].FQ9999A := 0.0;
results[i].FQ9999B := 0.0;
results[i].FQ9999C := 0.0;
results[i].FT9999Aavg := 0.0;
results[i].FT9999Bavg := 0.0;
results[i].FT9999Cavg := 0.0;
IF pumpA THEN
	results[i].P9999Arpm := sp[i];
	results[i].P9999Brpm := 0.0;
	MAIN.P9999A.nRun_RQ := 1; //start pump
	MAIN.P9999A.fSpeedSP_RQ := sp[i];
	MAIN.P9999B.nRun_RQ := 0; //stop pump
	MAIN.P9999B.fSpeedSP_RQ := 0.0;
ELSE
	results[i].P9999Arpm := 0.0;
	results[i].P9999Brpm := sp[i];
	MAIN.P9999A.nRun_RQ := 0; //stop pump
	MAIN.P9999A.fSpeedSP_RQ := 0.0;
	MAIN.P9999B.nRun_RQ := 1; //start pump
	MAIN.P9999B.fSpeedSP_RQ := sp[i];
END_IF
results[i].P9999Atubing := MAIN.P9999A.nTubeSize;
results[i].P9999Btubing := MAIN.P9999B.nTubeSize;
END_ACTION

ACTION recordTest_entry:
results[i].FQ9999A := MAIN.fbFQ9999A.total;
results[i].FQ9999B := MAIN.fbFQ9999B.total;
results[i].FQ9999C := MAIN.fbFQ9999C.total;
t := DWORD_TO_LREAL(TIME_TO_DWORD(runTestDuration))/1000.0/60.0;
results[i].FT9999Aavg := MAIN.fbFQ9999A.total/t;
results[i].FT9999Bavg := MAIN.fbFQ9999B.total/t;
results[i].FT9999Cavg := MAIN.fbFQ9999C.total/t;
END_ACTION

ACTION Init_entry:
IF i >= n THEN
	MAIN.P9999A.nRun_RQ := 0; //stop pump
	MAIN.P9999B.nRun_RQ := 0; //stop pump
	start := FALSE;
	i := 0;
END_IF
END_ACTION

END_PROGRAM

// ---- POUs/SonotecFreq.TcPOU
FUNCTION_BLOCK SonotecFreq
VAR_INPUT
	rawCount  AT %I* : UDINT;
	scale : sEU_SCALE := (rawLo := 0, rawHi := 20, euLo := -20.0,  euHi := 500.0, eu := 'ml/min');
END_VAR
VAR_OUTPUT
	pv : LREAL;
END_VAR
VAR
	lastCount : UDINT := 0;
	thisCount : INT;
END_VAR

thisCount := UDINT_TO_INT(rawCount - lastCount);
lastcount := rawCount;

SonotecFreq.pv := scale.euLo + (thisCount - scale.rawLo)*(scale.euHi - scale.euLo)/(scale.rawHi - scale.rawLo);

END_FUNCTION_BLOCK

// ---- POUs/Wiesler/AO1.TcPOU
FUNCTION_BLOCK AO1
VAR_INPUT
	out : LREAL;
	rawStatus : INT;
	scale : sEU_SCALE;
	sim : sAnalogSim;
END_VAR
VAR_OUTPUT
	rawOut : INT := 0;
END_VAR
VAR
END_VAR

IF sim.simEnable THEN
	rawOut := scale.rawLo + LREAL_TO_INT((sim.simValue - scale.euLo)*(scale.rawHi - scale.rawLo)/(scale.euHi - scale.euLo));
ELSE
	rawOut := scale.rawLo + LREAL_TO_INT((out - scale.euLo)*(scale.rawHi - scale.rawLo)/(scale.euHi - scale.euLo));
END_IF

END_FUNCTION_BLOCK

// ---- POUs/Wiesler/Datalog/fbDatalogger_1s.TcPOU
FUNCTION_BLOCK fbDatalogger_1s

VAR CONSTANT
	nRate : DINT := 1000;
	nPoints : DINT := 1000 / nRate;
END_VAR

VAR_INPUT
	fData : LREAL;
END_VAR
VAR_OUTPUT
	afLog : ARRAY[0..(nPoints-1)] OF LREAL;
	nLogJSTime : ULINT := 0;
END_VAR
VAR
	afCache : ARRAY[0..(nPoints-1)] OF LREAL;
	nCount : DINT := 0;
END_VAR

IF unixTime MOD DINT_TO_ULINT(nRate) = 0 THEN
	// Fill up the SampleArray
	afCache[nCount] := fData;
	// Increase the sampleIndex
	nCount := nCount + 1;
END_IF

IF nCount >= nPoints THEN
	// Copy values into log array
	afLog := afCache;
	// Increment log index to tell watching external logger the data has changed
	nLogJSTime := unixTime;
	// Reset count
	nCount := 0;
END_IF

END_FUNCTION_BLOCK

// ---- POUs/Wiesler/Datalog/fbDatalogger_20ms.TcPOU
FUNCTION_BLOCK fbDatalogger_20ms

VAR CONSTANT
	nRate : DINT := 20;
	nPoints : DINT := 1000 / nRate;
END_VAR

VAR_INPUT
	fData : LREAL;
END_VAR
VAR_OUTPUT
	afLog : ARRAY[0..(nPoints-1)] OF LREAL;
	nLogJSTime : ULINT := 0;
END_VAR
VAR
	afCache : ARRAY[0..(nPoints-1)] OF LREAL;
	nCount : DINT := 0;
END_VAR

IF unixTime MOD DINT_TO_ULINT(nRate) = 0 THEN
	// Fill up the SampleArray
	afCache[nCount] := fData;
	// Increase the sampleIndex
	nCount := nCount + 1;
END_IF

IF nCount >= nPoints THEN
	// Copy values into log array
	afLog := afCache;
	// Increment log index to tell watching external logger the data has changed
	nLogJSTime := unixTime;
	// Reset count
	nCount := 0;
END_IF

END_FUNCTION_BLOCK

// ---- POUs/Wiesler/fbDatalogger.TcPOU
FUNCTION_BLOCK fbDatalogger
VAR_INPUT
	fData : LREAL;
END_VAR
VAR_OUTPUT
	afLog : ARRAY[0..999] OF LREAL;
	nLogJSTime : ULINT := 0;
END_VAR
VAR
	afCache : ARRAY[0..999] OF LREAL;
	nCount : DINT := 0;
	nPoints : DINT := 1000;
END_VAR

// Fill up the SampleArray
afCache[nCount] := fData;
// Increase the sampleIndex
nCount := nCount + 1;
IF nCount >= nPoints THEN
	// Copy values into log array
	afLog := afCache;
	// Increment log index to tell watching external logger the data has changed
	nLogJSTime := unixTime;
	// Reset count
	nCount := 0;
END_IF

END_FUNCTION_BLOCK

// ---- POUs/Wiesler/FlowConcentrationControl/FlowSequence_CC1Test.TcPOU
PROGRAM FlowSequence_CC1Test
VAR_INPUT
	start : BOOL := FALSE;
	setSpeedDuration : TIME := T#15S;
	runTestDuration : TIME := T#2M;
	autoAdvance : BOOL := TRUE;
END_VAR
VAR_OUTPUT
	startTimes : ARRAY[1..50] OF ULINT;
	endTimes : ARRAY[1..50] OF ULINT;

	P9999Atubing : ARRAY[1..50] OF INT;
	P9999Btubing : ARRAY[1..50] OF INT;
END_VAR
VAR
	i : UINT := 0; // index
	n : UINT := 25;
	t : LREAL := 0.0;
	tol : LREAL := 5.0;
	spTotal : ARRAY [1..50] OF LREAL := [100.0,100.0,100.0,0.0,0.0,0.0,0.0,0.0,0.0,0.0,0.0,0.0,0.0,0.0,0.0,0.0,0.0,0.0,0.0,0.0,0.0,0.0,0.0,0.0, 0.0,
									0.0,0.0,0.0,0.0,0.0,0.0,0.0,0.0,0.0,0.0,0.0,0.0,0.0,0.0,0.0,0.0,0.0,0.0,0.0,0.0,0.0,0.0,0.0,0.0,0.0];
	//spTotal : ARRAY [1..50] OF LREAL := [100.0, 150.0, 200.0, 300.0, 150.0, 100.0, 80.0, 80.0, 90.0, 100.0, 
    //                                110.0, 120.0, 130.0, 140.0, 150.0, 0.0, 0.0, 0.0,
    //                                0.0, 0.0, 0.0, 0.0, 0.0, 0.0,
	//								0.0,0.0,0.0,0.0,0.0,0.0,0.0,0.0,0.0,0.0,0.0,0.0,0.0,0.0,0.0,0.0,0.0,0.0,0.0,0.0,0.0,0.0,0.0,0.0];
	spConc : ARRAY [1..50] OF LREAL := [1.0, 1.0, 1.0, 1.0, 1.0, 1.0, 1.0, 1.0, 1.0, 1.0, 
                                    1.0, 1.0, 1.0, 1.0, 1.0, 0.0, 0.0, 0.0,
                                    0.0, 0.0, 0.0, 0.0, 0.0, 0.0,
									0.0,0.0,0.0,0.0,0.0,0.0,0.0,0.0,0.0,0.0,0.0,0.0,0.0,0.0,0.0,0.0,0.0,0.0,0.0,0.0,0.0,0.0,0.0,0.0];
	
	setSpeed : SFCStepType;
	runTest : SFCStepType;
	recordTest : SFCStepType;
END_VAR

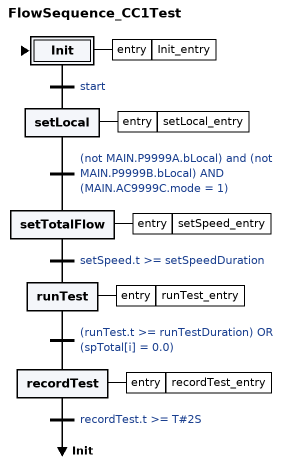
INITIAL_STEP Init:
    Init_entry(P1);  // entry action
END_STEP
TRANSITION FROM Init TO setLocal
    := start;
END_TRANSITION
STEP setLocal:
    setLocal_entry(P1);  // entry action
END_STEP
TRANSITION FROM setLocal TO setTotalFlow
    := (not MAIN.P9999A.bLocal) and (not MAIN.P9999B.bLocal) AND (MAIN.AC9999C.mode = 1);
END_TRANSITION
STEP setTotalFlow:
    setSpeed_entry(P1);  // entry action
END_STEP
TRANSITION FROM setTotalFlow TO runTest
    := setSpeed.t >= setSpeedDuration;
END_TRANSITION
STEP runTest:
    runTest_entry(P1);  // entry action
END_STEP
TRANSITION FROM runTest TO recordTest
    := (runTest.t >= runTestDuration) OR (spTotal[i] = 0.0);
END_TRANSITION
STEP recordTest:
    recordTest_entry(P1);  // entry action
END_STEP
TRANSITION FROM recordTest TO Init
    := recordTest.t >= T#2S;
END_TRANSITION

ACTION setLocal_entry:
IF MAIN.P9999A.bLocal THEN
	MAIN.P9999A.nLocal_RQ := 0;  //put pump in remote
END_IF
IF MAIN.P9999B.bLocal THEN
	MAIN.P9999B.nLocal_RQ := 0;  //put pump in remote
END_IF

IF MAIN.AC9999C.mode <> 1 THEN // concentration control in auto
	MAIN.AC9999C.c.rq := 0; // set initial total flow
	MAIN.AC9999C.conc.rq := 1.0; // set initial concentration
	MAIN.AC9999C.mode := 1;
END_IF
END_ACTION

ACTION Init_entry:
IF i >= n THEN
	MAIN.AC9999C.mode := 0; // concentration control in manual
	MAIN.P9999A.nRun_RQ := 0; //stop pump
	MAIN.P9999B.nRun_RQ := 0; //stop pump
	start := FALSE;
	i := 0;
END_IF
MAIN.logActive := FALSE;
END_ACTION

ACTION resetTotals_entry:
MAIN.fbFQ9999A.resetRQ := TRUE;
MAIN.fbFQ9999B.resetRQ := TRUE;
MAIN.fbFQ9999C.resetRQ := TRUE;
MAIN.MTSendString := 'ZI$0D$0A';
MAIN.logActive := TRUE;
END_ACTION

ACTION runTest_entry:
MAIN.MTSendString := 'SIR$0D$0A';
startTimes[i] := unixTime;
END_ACTION

ACTION setSpeed_entry:
i := i + 1;
startTimes[i] := 0;
endTimes[i] := 0;

MAIN.AC9999C.c.rq := spTotal[i];
MAIN.AC9999C.conc.rq := spConc[i];

P9999Atubing[i] := MAIN.P9999A.nTubeSize;
P9999Btubing[i] := MAIN.P9999B.nTubeSize;
END_ACTION

ACTION recordTest_entry:
endTimes[i] := unixTime;

t := DWORD_TO_LREAL(TIME_TO_DWORD(runTestDuration))/1000.0/60.0;

IF NOT autoAdvance THEN
	start := FALSE;
END_IF
END_ACTION

END_PROGRAM

// ---- GlobalTextList.TcGTLO
TEXTLIST GlobalTextList
  23 = '%.1f'
  9 = '%.3f'
  12 = 'ABS 300: %.3f'
  11 = 'ABS 313: %.3f'
  13 = 'ABSDELTA: %.3f'
  5 = 'API'
  3 = 'API Flow: %3.2f mg/min'
  1 = 'API Flow: %f mg/min'
  2 = 'API Flow: %f3.2 mg/min'
  0 = 'API Flow: %r mg/min'
  7 = 'Aseptic Filter'
  20 = 'AT'
  4 = 'Buffer'
  10 = 'CONC:  %.1f'
  8 = 'Filler'
  19 = 'FT'
  21 = 'INPUT'
  6 = 'OOS'
  18 = 'PT'
  25 = 'PV:  %.1f RPM'
  14 = 'Reveal 290: %.3f'
  15 = 'Reveal 300: %.3f'
  16 = 'Reveal 310: %.3f'
  17 = 'Reveal 320: %.3f'
  24 = 'SP: %.1f RPM'
  22 = 'Speed SP'
END_TEXTLIST

// ---- VISUs/ContinuousFormulation.TcVIS
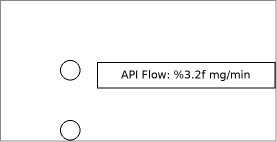
VISUALIZATION ContinuousFormulation  // 277x142
    Ellipse (60,60 20x20)
    Ellipse (60,120 20x20)
    Rectangle (97,62 178x26), "API Flow: %3.2f mg/min", text variable: IO.FT_API_PV
END_VISUALIZATION

